METHOD FB_init : BOOL
VAR_INPUT
	bInitRetains : BOOL; // if TRUE, the retain variables are initialized (warm start / cold start)
	bInCopyCode : BOOL;  // if TRUE, the instance afterwards gets moved into the copy code (online change)
END_VAR
AddInput('ipSrcImage', ipSrcImage);
AddInput('ipTemplateImage', ipTemplateImage);
AddInput('fMatchThreshold', fMatchThreshold);
AddInput('nProjections', nProjections);
AddInput('eOptions', eOptions);
AddInput('nRotations', nRotations);
AddInput('fScaleFactor', fScaleFactor);
AddInput('eInterpolationType', eInterpolationType);
AddInput('hrPrev', hrPrev);
AddOutput('ipMatches', ipMatches);
AddOutput('ipMatchValues', ipMatchValues);
AddOutput('hresult',hresult);
END_METHOD

METHOD PUBLIC  Clone : I_Node
VAR
	pNode : POINTER TO Node_F_VN_FindTemplateWalshExp;
END_VAR
pNode := __NEW(Node_F_VN_FindTemplateWalshExp);
Clone := pNode^;
END_METHOD

METHOD PROTECTED OnExecute
hresult.Value := F_VN_FindTemplateWalshExp(
    ipSrcImage := ipSrcImage.Value,
    ipTemplateImage := ipTemplateImage.Value,
	ipMatches := ipMatches.Value,
	fMatchThreshold := fMatchThreshold.Value,
	nProjections := nProjections.Value,
	eOptions := eOptions.Value,
	nRotations := nRotations.Value,
	fScaleFactor := fScaleFactor.Value,
	eInterpolationType := eInterpolationType.Value,
	ipMatchValues := ipMatchValues.Value,
	hrPrev:= hrPrev.Value);
END_METHOD

METHOD PUBLIC PreExecutionCheck
VAR_INPUT
	Check : I_PreExecutionChecks;
END_VAR
Check.IsTrue(ipSrcImage.IsValid, 'ipSrcImage must contain an image');
Check.IsTrue(ipSrcImage.IsPixelDepth(8), 'ipSrcImage must be 8 or 32 bit pixel depth');
Check.IsTrue((ipSrcImage.HasChannelCount(1) OR ipSrcImage.HasChannelCount(3)), 'ipSrcImage must contain 1 or 3 channels');

Check.IsTrue((nRotations.Value = 1 OR nRotations.Value = 2 OR nRotations.Value = 4 OR nRotations.Value = 8 OR nRotations.Value = 16 OR nRotations.Value = 32), 'nRotations must be 1, 2, 4, 8, 16 or 32');
Check.IsTrue((fMatchThreshold.Value >= 0 AND fMatchThreshold.Value <= 1), 'Threshold must be between 0..1, 1.0 would be a perfect match');
Check.IsTrue(nProjections.Value <= 50, 'The soft limit of 50 has been reached');

Check.IsTrue(ipTemplateImage.IsValid, 'ipTemplateImage must contain an image');
Check.IsTrue(ImagesHaveMatchingPixelFormats(ipSrcImage.Value, ipTemplateImage.Value), 'ipTemplateImage must have same pixel depth as ipSrcImage');
Check.IsTrue(ImagesHaveMatchingChannels(ipSrcImage.Value, ipTemplateImage.Value), 'ipTemplateImage must have same amount of channels as ipSrcImage');
Check.IsTrue(IsTemplateImageSmallerThanSourceImage(ipSrcImage.Value, ipTemplateImage.Value), 'ipTemplateImage must be smaller than ipSrcImage');
END_METHOD

END_FUNCTION_BLOCK

// Nodes/Image Analysis/Object Detection/Node_F_VN_FindTemplateWalshExp_AngleRange
{attribute 'linkalways'} 
{attribute 'no_explicit_call' := 'This FB is a CLASS and must be accessed using methods or properties'}
{attribute 'enable_dynamic_creation'}
FUNCTION_BLOCK Node_F_VN_FindTemplateWalshExp_AngleRange EXTENDS VisionNode
VAR
    ipSrcImage : _ITcVnImage;
    ipTemplateImage : _ITcVnImage;
	ipMatches : _ITcVnContainer;
	fMatchThreshold : _REAL(0.1);
	nProjections : _UDINT(10);
	fStartAngle : _LREAL(0);
	fStopAngle : _LREAL(1);
	nAngles : _UDINT(1);
	eOptions : _ETcVnFindTemplateWalshOptions(ETcVnFindTemplateWalshOptions.TCVN_FTWO_NONE);
	fScaleFactor : _REAL(1);
	eInterpolationType : _ETcVnInterpolationType(ETcVnInterpolationType.TCVN_IT_AREA_BASED);
	ipMatchValues : _ITcVnContainer;
    hrPrev : _HRESULT(S_OK);
	hresult : _HRESULT(S_OK);
END_VAR

METHOD FB_init : BOOL
VAR_INPUT
	bInitRetains : BOOL; // if TRUE, the retain variables are initialized (warm start / cold start)
	bInCopyCode : BOOL;  // if TRUE, the instance afterwards gets moved into the copy code (online change)
END_VAR
AddInput('ipSrcImage', ipSrcImage);
AddInput('ipTemplateImage', ipTemplateImage);
AddInput('fMatchThreshold', fMatchThreshold);
AddInput('nProjections', nProjections);
AddInput('fStartAngle', fStartAngle);
AddInput('fStopAngle', fStopAngle);
AddInput('nAngles', nAngles);
AddInput('eOptions', eOptions);
AddInput('fScaleFactor', fScaleFactor);
AddInput('eInterpolationType', eInterpolationType);
AddInput('hrPrev', hrPrev);
AddOutput('ipMatches', ipMatches);
AddOutput('ipMatchValues', ipMatchValues);
AddOutput('hresult',hresult);
END_METHOD

METHOD PUBLIC  Clone : I_Node
VAR
	pNode : POINTER TO Node_F_VN_FindTemplateWalshExp_AngleRange;
END_VAR
pNode := __NEW(Node_F_VN_FindTemplateWalshExp_AngleRange);
Clone := pNode^;
END_METHOD

METHOD PROTECTED OnExecute
hresult.Value := F_VN_FindTemplateWalshExp_AngleRange(
    ipSrcImage := ipSrcImage.Value,
    ipTemplateImage := ipTemplateImage.Value,
	ipMatches := ipMatches.Value,
	fMatchThreshold := fMatchThreshold.Value,
	nProjections := nProjections.Value,
	fStartAngle := fStartAngle.Value,
	fStopAngle := fStopAngle.Value,
	nAngles := nAngles.Value,
	eOptions := eOptions.Value,
	fScaleFactor := fScaleFactor.Value,
	eInterpolationType := eInterpolationType.Value,
	ipMatchValues := ipMatchValues.Value,
	hrPrev:= hrPrev.Value);
END_METHOD

METHOD PUBLIC PreExecutionCheck
VAR_INPUT
	Check : I_PreExecutionChecks;
END_VAR
Check.IsTrue(ipSrcImage.IsValid, 'ipSrcImage must contain an image');
Check.IsTrue(ipSrcImage.IsPixelDepth(8), 'ipSrcImage must be 8 or 32 bit pixel depth');
Check.IsTrue((ipSrcImage.HasChannelCount(1) OR ipSrcImage.HasChannelCount(3)), 'ipSrcImage must contain 1 or 3 channels');

Check.IsTrue((fMatchThreshold.Value >= 0 AND fMatchThreshold.Value <= 1), 'Threshold must be between 0..1, 1.0 would be a perfect match');
Check.IsTrue(nProjections.Value <= 50, 'The soft limit of 50 has been reached');

Check.IsTrue(ipTemplateImage.IsValid, 'ipTemplateImage must contain an image');
Check.IsTrue(ImagesHaveMatchingPixelFormats(ipSrcImage.Value, ipTemplateImage.Value), 'ipTemplateImage must have same pixel depth as ipSrcImage');
Check.IsTrue(ImagesHaveMatchingChannels(ipSrcImage.Value, ipTemplateImage.Value), 'ipTemplateImage must have same amount of channels as ipSrcImage');
Check.IsTrue(IsTemplateImageSmallerThanSourceImage(ipSrcImage.Value, ipTemplateImage.Value), 'ipTemplateImage must be smaller than ipSrcImage');
END_METHOD

END_FUNCTION_BLOCK

// Nodes/Image Analysis/Object Detection/Node_F_VN_HoughCircles
{attribute 'linkalways'} 
{attribute 'no_explicit_call' := 'This FB is a CLASS and must be accessed using methods or properties'}
{attribute 'enable_dynamic_creation'}
FUNCTION_BLOCK Node_F_VN_HoughCircles EXTENDS VisionNode
VAR
    ipSrcImage : _ITcVnImage;
    ipCircles : _ITcVnContainer;
    fInvAccuRatio : _LREAL(1.0);
    fMinDist : _LREAL(1.0);
    hrPrev : _HRESULT(S_OK);
	hresult : _HRESULT(S_OK);
END_VAR

METHOD FB_init : BOOL
VAR_INPUT
	bInitRetains : BOOL; // if TRUE, the retain variables are initialized (warm start / cold start)
	bInCopyCode : BOOL;  // if TRUE, the instance afterwards gets moved into the copy code (online change)
END_VAR
AddInput('ipSrcImage', ipSrcImage);
AddParameter('fInvAccuRatio', fInvAccuRatio);
AddParameter('fMinDist', fMinDist);
AddInput('hrPrev', hrPrev);
AddOutput('ipCircles', ipCircles);
AddOutput('hresult', hresult);
END_METHOD

METHOD PUBLIC  Clone : I_Node
VAR
	pNode : POINTER TO Node_F_VN_HoughCircles;
END_VAR
pNode := __NEW(Node_F_VN_HoughCircles);
Clone := pNode^;
END_METHOD

METHOD PROTECTED OnExecute
hresult.Value := F_VN_HoughCircles(
	ipSrcImage := ipSrcImage.Value,
    ipCircles := ipCircles.Value,
    fInvAccuRatio := fInvAccuRatio.Value,
    fMinDist := fMinDist.Value,
	hrPrev:= hrPrev.Value);
END_METHOD

METHOD PUBLIC PreExecutionCheck
VAR_INPUT
	Check : I_PreExecutionChecks;
END_VAR
Check.IsTrue(ipSrcImage.IsValid, 'ipSrcImage must contain an image');
Check.IsTrue(ipSrcImage.IsElementType(ETcVnElementType.TCVN_ET_USINT), 'ipSrcImage must be usint');
Check.IsTrue(ipSrcImage.HasChannelCount(1), 'ipSrcImage must contain 1 channel');
Check.IsTrue((fInvAccuRatio.Value > 0), 'fInvAccuRatio must be greater than 0');
Check.IsTrue((fMinDist.Value > 0), 'fMinDist must be greater than 0');
END_METHOD

END_FUNCTION_BLOCK

// Nodes/Image Analysis/Object Detection/Node_F_VN_HoughCirclesExp
{attribute 'linkalways'} 
{attribute 'no_explicit_call' := 'This FB is a CLASS and must be accessed using methods or properties'}
{attribute 'enable_dynamic_creation'}
FUNCTION_BLOCK Node_F_VN_HoughCirclesExp EXTENDS VisionNode
VAR
    ipSrcImage : _ITcVnImage;
    ipCircles : _ITcVnContainer;
    fInvAccuRatio : _LREAL(1.0);
    fMinDist : _LREAL(1.0);
	eHoughMethod : _ETcVnHoughMethod(ETcVnHoughMethod.TCVN_HM_GRADIENT);
    fParam1 : _LREAL(0.0);
	fParam2 : _LREAL(0.0);
	nMinRadius : _UDINT(0);
	nMaxRadius : _UDINT(0);
	hrPrev : _HRESULT(S_OK);
	hresult : _HRESULT(S_OK);
END_VAR

METHOD FB_init : BOOL
VAR_INPUT
	bInitRetains : BOOL; // if TRUE, the retain variables are initialized (warm start / cold start)
	bInCopyCode : BOOL;  // if TRUE, the instance afterwards gets moved into the copy code (online change)
END_VAR
AddInput('ipSrcImage', ipSrcImage);
AddParameter('fInvAccuRatio', fInvAccuRatio);
AddParameter('fMinDist', fMinDist);
AddParameter('eHoughMethod', eHoughMethod);
AddParameter('fParam1', fParam1);
AddParameter('fParam2', fParam2);
AddParameter('nMinRadius', nMinRadius);
AddParameter('nMaxRadius', nMaxRadius);
AddInput('hrPrev', hrPrev);
AddOutput('ipCircles', ipCircles);
AddOutput('hresult', hresult);
END_METHOD

METHOD PUBLIC  Clone : I_Node
VAR
	pNode : POINTER TO Node_F_VN_HoughCirclesExp;
END_VAR
pNode := __NEW(Node_F_VN_HoughCirclesExp);
Clone := pNode^;
END_METHOD

METHOD PROTECTED OnExecute
hresult.Value := F_VN_HoughCirclesExp(
	ipSrcImage := ipSrcImage.Value,
    ipCircles := ipCircles.Value,
    fInvAccuRatio := fInvAccuRatio.Value,
    fMinDist := fMinDist.Value,
	eHoughMethod := eHoughMethod.Value,
	fParam1 := fParam1.Value,
	fParam2 := fParam2.Value,
	nMinRadius := nMinRadius.Value,
	nMaxRadius := nMaxRadius.Value,
	hrPrev:= hrPrev.Value);
END_METHOD

METHOD PUBLIC PreExecutionCheck
VAR_INPUT
	Check : I_PreExecutionChecks;
END_VAR
Check.IsTrue(ipSrcImage.IsValid, 'ipSrcImage must contain an image');
Check.IsTrue(ipSrcImage.IsElementType(ETcVnElementType.TCVN_ET_USINT), 'ipSrcImage must be usint');
Check.IsTrue(ipSrcImage.HasChannelCount(1), 'ipSrcImage must contain 1 channel');
Check.IsTrue((fInvAccuRatio.Value > 0), 'fInvAccuRatio must be greater than 0');
Check.IsTrue((fMinDist.Value > 0), 'fMinDist must be greater than 0');

Check.IsTrue(
    (eHoughMethod.Value = ETcVnHoughMethod.TCVN_HM_GRADIENT) OR
    (eHoughMethod.Value = ETcVnHoughMethod.TCVN_HM_GRADIENT_ALT),
    'eHoughMethod must be GRADIENT or GRADIENT_ALT');
	
	
IF (eHoughMethod.Value = ETcVnHoughMethod.TCVN_HM_GRADIENT_ALT) THEN
    Check.IsTrue((fParam2.Value > 0) AND (fParam2.Value < 1),
        'fParam2 (circle perfectness) must be > 0 and < 1 for GRADIENT_ALT');
ELSE
    Check.IsTrue((fParam2.Value > 0),
        'fParam2 (accumulator threshold) must be > 0 for GRADIENT');
END_IF

IF (nMaxRadius.Value > 0) THEN
    Check.IsTrue((nMaxRadius.Value >= nMinRadius.Value),
        'nMaxRadius must be >= nMinRadius when non-zero');
END_IF
END_METHOD

END_FUNCTION_BLOCK

// Nodes/Image Analysis/Object Detection/Node_F_VN_HoughLines
{attribute 'linkalways'} 
{attribute 'no_explicit_call' := 'This FB is a CLASS and must be accessed using methods or properties'}
{attribute 'enable_dynamic_creation'}
FUNCTION_BLOCK Node_F_VN_HoughLines EXTENDS VisionNode
VAR
    ipSrcImage : _ITcVnImage;
    ipLines : _ITcVnContainer;
    fDistRes : _LREAL(1.0);
    fAngleRes : _LREAL(1.0);
    nAccuThreshold : _UDINT(0);
    hrPrev : _HRESULT(S_OK);
	hresult : _HRESULT(S_OK);
END_VAR

METHOD FB_init : BOOL
VAR_INPUT
	bInitRetains : BOOL; // if TRUE, the retain variables are initialized (warm start / cold start)
	bInCopyCode : BOOL;  // if TRUE, the instance afterwards gets moved into the copy code (online change)
END_VAR
AddInput('ipSrcImage', ipSrcImage);
AddParameter('fDistRes', fDistRes);
AddParameter('fAngleRes', fAngleRes);
AddParameter('nAccuThreshold', nAccuThreshold);
AddInput('hrPrev', hrPrev);
AddOutput('ipLines', ipLines);
AddOutput('hresult', hresult);
END_METHOD

METHOD PUBLIC  Clone : I_Node
VAR
	pNode : POINTER TO Node_F_VN_HoughLines;
END_VAR
pNode := __NEW(Node_F_VN_HoughLines);
Clone := pNode^;
END_METHOD

METHOD PROTECTED OnExecute
hresult.Value := F_VN_HoughLines(
	ipSrcImage := ipSrcImage.Value,
    ipLines := ipLines.Value,
    fDistRes := fDistRes.Value,
    fAngleRes := fAngleRes.Value,
    nAccuThreshold := nAccuThreshold.Value,
	hrPrev:= hrPrev.Value);
END_METHOD

METHOD PUBLIC PreExecutionCheck
VAR_INPUT
	Check : I_PreExecutionChecks;
END_VAR
Check.IsTrue(ipSrcImage.IsValid, 'ipSrcImage must contain an image');
Check.IsTrue(ipSrcImage.IsPixelDepth(8), 'ipSrcImage must be 8 bit pixel depth');
Check.IsTrue(ipSrcImage.HasChannelCount(1), 'ipSrcImage must contain 1 channel');
Check.IsTrue((fDistRes.Value > 0), 'fDistRes must be greater than 0');
Check.IsTrue((fAngleRes.Value > 0), 'fAngleRes must be greater than 0');
END_METHOD

END_FUNCTION_BLOCK

// Nodes/Image Analysis/Object Detection/Node_F_VN_HoughLinesP
{attribute 'linkalways'} 
{attribute 'no_explicit_call' := 'This FB is a CLASS and must be accessed using methods or properties'}
{attribute 'enable_dynamic_creation'}
FUNCTION_BLOCK Node_F_VN_HoughLinesP EXTENDS VisionNode
VAR
    ipSrcImage : _ITcVnImage;
    ipLines : _ITcVnContainer;
    fDistRes : _LREAL(1.0);
    fAngleRes : _LREAL(1.0);
    nAccuThreshold : _UDINT(0);
    hrPrev : _HRESULT(S_OK);
	hresult : _HRESULT(S_OK);
END_VAR

METHOD FB_init : BOOL
VAR_INPUT
	bInitRetains : BOOL; // if TRUE, the retain variables are initialized (warm start / cold start)
	bInCopyCode : BOOL;  // if TRUE, the instance afterwards gets moved into the copy code (online change)
END_VAR
AddInput('ipSrcImage', ipSrcImage);
AddParameter('fDistRes', fDistRes);
AddParameter('fAngleRes', fAngleRes);
AddParameter('nAccuThreshold', nAccuThreshold);
AddInput('hrPrev', hrPrev);
AddOutput('ipLines', ipLines);
AddOutput('hresult', hresult);
END_METHOD

METHOD PUBLIC  Clone : I_Node
VAR
	pNode : POINTER TO Node_F_VN_HoughLinesP;
END_VAR
pNode := __NEW(Node_F_VN_HoughLinesP);
Clone := pNode^;
END_METHOD

METHOD PROTECTED OnExecute
hresult.Value := F_VN_HoughLinesP(
	ipSrcImage := ipSrcImage.Value,
    ipLines := ipLines.Value,
    fDistRes := fDistRes.Value,
    fAngleRes := fAngleRes.Value,
    nAccuThreshold := nAccuThreshold.Value,
	hrPrev:= hrPrev.Value);
END_METHOD

METHOD PUBLIC PreExecutionCheck
VAR_INPUT
	Check : I_PreExecutionChecks;
END_VAR
Check.IsTrue(ipSrcImage.IsValid, 'ipSrcImage must contain an image');
Check.IsTrue(ipSrcImage.IsPixelDepth(8), 'ipSrcImage must be 8 bit pixel depth');
Check.IsTrue(ipSrcImage.HasChannelCount(1), 'ipSrcImage must contain 1 channel');
Check.IsTrue((fDistRes.Value > 0), 'fDistRes must be greater than 0');
Check.IsTrue((fAngleRes.Value > 0), 'fAngleRes must be greater than 0');
END_METHOD

END_FUNCTION_BLOCK

// Nodes/Image Analysis/Object Detection/Node_F_VN_HoughLinesPExp
{attribute 'linkalways'} 
{attribute 'no_explicit_call' := 'This FB is a CLASS and must be accessed using methods or properties'}
{attribute 'enable_dynamic_creation'}
FUNCTION_BLOCK Node_F_VN_HoughLinesPExp EXTENDS VisionNode
VAR
    ipSrcImage : _ITcVnImage;
    ipLines : _ITcVnContainer;
    fDistRes : _LREAL(1.0);
    fAngleRes : _LREAL(1.0);
    nAccuThreshold : _UDINT(0);
    fMinLineLength : _LREAL(0.0);
    fMaxLineGap : _LREAL(0.0);
    hrPrev : _HRESULT(S_OK);
	hresult : _HRESULT(S_OK);
END_VAR

METHOD FB_init : BOOL
VAR_INPUT
	bInitRetains : BOOL; // if TRUE, the retain variables are initialized (warm start / cold start)
	bInCopyCode : BOOL;  // if TRUE, the instance afterwards gets moved into the copy code (online change)
END_VAR
AddInput('ipSrcImage', ipSrcImage);
AddParameter('fDistRes', fDistRes);
AddParameter('fAngleRes', fAngleRes);
AddParameter('nAccuThreshold', nAccuThreshold);
AddParameter('fMinLineLength', fMinLineLength);
AddParameter('fMaxLineGap', fMaxLineGap);
AddInput('hrPrev', hrPrev);
AddOutput('ipLines', ipLines);
AddOutput('hresult', hresult);
END_METHOD

METHOD PUBLIC  Clone : I_Node
VAR
	pNode : POINTER TO Node_F_VN_HoughLinesPExp;
END_VAR
pNode := __NEW(Node_F_VN_HoughLinesPExp);
Clone := pNode^;
END_METHOD

METHOD PROTECTED OnExecute
hresult.Value := F_VN_HoughLinesPExp(
	ipSrcImage := ipSrcImage.Value,
    ipLines := ipLines.Value,
    fDistRes := fDistRes.Value,
    fAngleRes := fAngleRes.Value,
    nAccuThreshold := nAccuThreshold.Value,
    fMinLineLength := fMinLineLength.Value,
    fMaxLineGap := fMaxLineGap.Value,
	hrPrev:= hrPrev.Value);
END_METHOD

METHOD PUBLIC PreExecutionCheck
VAR_INPUT
	Check : I_PreExecutionChecks;
END_VAR
Check.IsTrue(ipSrcImage.IsValid, 'ipSrcImage must contain an image');
Check.IsTrue(ipSrcImage.IsPixelDepth(8), 'ipSrcImage must be 8 bit pixel depth');
Check.IsTrue(ipSrcImage.HasChannelCount(1), 'ipSrcImage must contain 1 channel');
Check.IsTrue((fDistRes.Value > 0), 'fDistRes must be greater than 0');
Check.IsTrue((fAngleRes.Value > 0), 'fAngleRes must be greater than 0');
END_METHOD

END_FUNCTION_BLOCK

// Nodes/Image Analysis/Object Detection/Node_F_VN_MatchImageHuMoments
{attribute 'linkalways'} 
{attribute 'no_explicit_call' := 'This FB is a CLASS and must be accessed using methods or properties'}
{attribute 'enable_dynamic_creation'}
FUNCTION_BLOCK Node_F_VN_MatchImageHuMoments EXTENDS VisionNode
VAR
    ipImage1 : _ITcVnImage;
    ipImage2 : _ITcVnImage;
    eComparisonMethod : _ETcVnContoursMatchComparisonMethod(ETcVnContoursMatchComparisonMethod.TCVN_CMCM_CONTOURS_MATCH_I1);
    fDissimilarity : _LREAL(0.0);
    hrPrev : _HRESULT(S_OK);
	hresult : _HRESULT(S_OK);
END_VAR

METHOD FB_init : BOOL
VAR_INPUT
	bInitRetains : BOOL; // if TRUE, the retain variables are initialized (warm start / cold start)
	bInCopyCode : BOOL;  // if TRUE, the instance afterwards gets moved into the copy code (online change)
END_VAR
AddInput('ipImage1', ipImage1);
AddInput('ipImage2', ipImage2);
AddParameter('eComparisonMethod', eComparisonMethod);
AddInput('hrPrev', hrPrev);
AddOutput('fDissimilarity', fDissimilarity);
AddOutput('hresult', hresult);
END_METHOD

METHOD PUBLIC  Clone : I_Node
VAR
	pNode : POINTER TO Node_F_VN_MatchImageHuMoments;
END_VAR
pNode := __NEW(Node_F_VN_MatchImageHuMoments);
Clone := pNode^;
END_METHOD

METHOD PROTECTED OnExecute
hresult.Value := F_VN_MatchImageHuMoments(
	ipImage1 := ipImage1.Value,
    ipImage2 := ipImage2.Value,
    eComparisonMethod := eComparisonMethod.Value,
    fDissimilarity := fDissimilarity.Value,
	hrPrev:= hrPrev.Value);
END_METHOD

METHOD PUBLIC PreExecutionCheck
VAR_INPUT
	Check : I_PreExecutionChecks;
END_VAR
Check.IsTrue(ipImage1.IsValid, 'ipImage1 must contain an image');
Check.IsTrue(ipImage1.HasChannelCount(1), 'ipImage1 must contain 1 channel');
Check.IsTrue(ipImage2.IsValid, 'ipImage2 must contain an image');
Check.IsTrue(ipImage2.HasChannelCount(1), 'ipImage2 must contain 1 channel');
END_METHOD

END_FUNCTION_BLOCK

// Nodes/Image Analysis/Object Detection/Node_F_VN_MatchTemplate
{attribute 'linkalways'} 
{attribute 'no_explicit_call' := 'This FB is a CLASS and must be accessed using methods or properties'}
{attribute 'enable_dynamic_creation'}
FUNCTION_BLOCK Node_F_VN_MatchTemplate EXTENDS VisionNode
VAR
    ipSrcImage : _ITcVnImage;
    ipTemplateImage : _ITcVnImage;
    ipResultImage : _ITcVnImage;
    hrPrev : _HRESULT(S_OK);
	hresult : _HRESULT(S_OK);
END_VAR

METHOD FB_init : BOOL
VAR_INPUT
	bInitRetains : BOOL; // if TRUE, the retain variables are initialized (warm start / cold start)
	bInCopyCode : BOOL;  // if TRUE, the instance afterwards gets moved into the copy code (online change)
END_VAR
AddInput('ipSrcImage', ipSrcImage);
AddInput('ipTemplateImage', ipTemplateImage);
AddInput('hrPrev', hrPrev);
AddOutput('ipResultImage', ipResultImage);
AddOutput('hresult',hresult);
END_METHOD

METHOD PUBLIC  Clone : I_Node
VAR
	pNode : POINTER TO Node_F_VN_MatchTemplate;
END_VAR
pNode := __NEW(Node_F_VN_MatchTemplate);
Clone := pNode^;
END_METHOD

METHOD PROTECTED OnExecute
hresult.Value := F_VN_MatchTemplate(
    ipSrcImage := ipSrcImage.Value,
    ipTemplateImage := ipTemplateImage.Value,
	ipResultImage := ipResultImage.Value,
	hrPrev:= hrPrev.Value);
END_METHOD

METHOD PUBLIC PreExecutionCheck
VAR_INPUT
	Check : I_PreExecutionChecks;
END_VAR
Check.IsTrue(ipSrcImage.IsValid, 'ipSrcImage must contain an image');
Check.IsTrue((ipSrcImage.IsPixelDepth(8) OR ipSrcImage.IsPixelDepth(32)), 'ipSrcImage must be 8 or 32 bit pixel depth');
Check.IsTrue((ipSrcImage.HasChannelCount(1) OR ipSrcImage.HasChannelCount(3)), 'ipSrcImage must contain 1 or 3 channels');

Check.IsTrue(ipTemplateImage.IsValid, 'ipTemplateImage must contain an image');
Check.IsTrue(ImagesHaveMatchingPixelFormats(ipSrcImage.Value, ipTemplateImage.Value), 'ipTemplateImage must have same pixel depth as ipSrcImage');
Check.IsTrue(ImagesHaveMatchingChannels(ipSrcImage.Value, ipTemplateImage.Value), 'ipTemplateImage must have same amount of channels as ipSrcImage');
Check.IsTrue(IsTemplateImageSmallerThanSourceImage(ipSrcImage.Value, ipTemplateImage.Value), 'ipTemplateImage must be smaller than ipSrcImage');
END_METHOD

END_FUNCTION_BLOCK

// Nodes/Image Analysis/Object Detection/Node_F_VN_MatchTemplateAndEvaluate
{attribute 'linkalways'} 
{attribute 'no_explicit_call' := 'This FB is a CLASS and must be accessed using methods or properties'}
{attribute 'enable_dynamic_creation'}
FUNCTION_BLOCK Node_F_VN_MatchTemplateAndEvaluate EXTENDS VisionNode
VAR
    ipSrcImage : _ITcVnImage;
    ipTemplateImage : _ITcVnImage;
    ipMatches : _ITcVnContainer;
    fMatchThreshold : _REAL(0.0);
    hrPrev : _HRESULT(S_OK);
	hresult : _HRESULT(S_OK);
END_VAR

METHOD FB_init : BOOL
VAR_INPUT
	bInitRetains : BOOL; // if TRUE, the retain variables are initialized (warm start / cold start)
	bInCopyCode : BOOL;  // if TRUE, the instance afterwards gets moved into the copy code (online change)
END_VAR
AddInput('ipSrcImage', ipSrcImage);
AddInput('ipTemplateImage', ipTemplateImage);
AddParameter('fMatchThreshold', fMatchThreshold);
AddInput('hrPrev', hrPrev);
AddOutput('ipMatches', ipMatches);
AddOutput('hresult',hresult);
END_METHOD

METHOD PUBLIC  Clone : I_Node
VAR
	pNode : POINTER TO Node_F_VN_MatchTemplateAndEvaluate;
END_VAR
pNode := __NEW(Node_F_VN_MatchTemplateAndEvaluate);
Clone := pNode^;
END_METHOD

METHOD PROTECTED OnExecute
hresult.Value := F_VN_MatchTemplateAndEvaluate(
    ipSrcImage := ipSrcImage.Value,
    ipTemplateImage := ipTemplateImage.Value,
	ipMatches := ipMatches.Value,
    fMatchThreshold := fMatchThreshold.Value,
	hrPrev:= hrPrev.Value);
END_METHOD

METHOD PUBLIC PreExecutionCheck
VAR_INPUT
	Check : I_PreExecutionChecks;
END_VAR
Check.IsTrue(ipSrcImage.IsValid, 'ipSrcImage must contain an image');
Check.IsTrue((ipSrcImage.IsPixelDepth(8) OR ipSrcImage.IsPixelDepth(32)), 'ipSrcImage must be 8 or 32 bit pixel depth');
Check.IsTrue((ipSrcImage.HasChannelCount(1) OR ipSrcImage.HasChannelCount(3)), 'ipSrcImage must contain 1 or 3 channels');

Check.IsTrue(ipTemplateImage.IsValid, 'ipTemplateImage must contain an image');
Check.IsTrue(ImagesHaveMatchingPixelFormats(ipSrcImage.Value, ipTemplateImage.Value), 'ipTemplateImage must have same pixel depth ipSrcImage');
Check.IsTrue(ImagesHaveMatchingChannels(ipSrcImage.Value, ipTemplateImage.Value), 'ipTemplateImage must have same amount of channels as ipSrcImage');
Check.IsTrue(IsTemplateImageSmallerThanSourceImage(ipSrcImage.Value, ipTemplateImage.Value), 'ipTemplateImage must be smaller than ipSrcImage');

Check.IsTrue((fMatchThreshold.Value >= 0.0) AND (fMatchThreshold.Value <= 1.0), 'fMatchThreshold must be between 0 and 1');
END_METHOD

END_FUNCTION_BLOCK

// Nodes/Image Analysis/Object Detection/Node_F_VN_MatchTemplateAndEvaluateExp
{attribute 'linkalways'}
{attribute 'no_explicit_call' := 'This FB is a CLASS and must be accessed using methods or properties'}
{attribute 'enable_dynamic_creation'}
FUNCTION_BLOCK Node_F_VN_MatchTemplateAndEvaluateExp EXTENDS VisionNode
VAR
    ipSrcImage : _ITcVnImage;
    ipTemplateImage : _ITcVnImage;
    ipMatches : _ITcVnContainer;
    fMatchThreshold : _REAL(0.0);
    eMatchMethod : _ETcVnTemplateMatchMethod(ETcVnTemplateMatchMethod.TCVN_TMM_CCORR_NORMED);
    ipTemplateMask : _ITcVnImage;
    fScaleFactor : _REAL(1);
    eInterpolationType : _ETcVnInterpolationType(ETcVnInterpolationType.TCVN_IT_BILINEAR);
    ipMatchValues : _ITcVnContainer;
    hrPrev : _HRESULT(S_OK);
    hresult : _HRESULT(S_OK);
END_VAR

METHOD FB_init : BOOL
VAR_INPUT
    bInitRetains : BOOL;
    bInCopyCode : BOOL;
END_VAR
AddInput('ipSrcImage', ipSrcImage);
AddInput('ipTemplateImage', ipTemplateImage);
AddOutput('ipMatches', ipMatches);
AddParameter('fMatchThreshold', fMatchThreshold);
AddParameter('eMatchMethod', eMatchMethod);
AddInput('ipTemplateMask', ipTemplateMask);
AddParameter('fScaleFactor', fScaleFactor);
AddParameter('eInterpolationType', eInterpolationType);
AddOutput('ipMatchValues', ipMatchValues);
AddInput('hrPrev', hrPrev);
AddOutput('hresult', hresult);
END_METHOD

METHOD PUBLIC Clone : I_Node
VAR
    pNode : POINTER TO Node_F_VN_MatchTemplateAndEvaluateExp;
END_VAR
pNode := __NEW(Node_F_VN_MatchTemplateAndEvaluateExp);
Clone := pNode^;
END_METHOD

METHOD PROTECTED OnExecute
hresult.Value := F_VN_MatchTemplateAndEvaluateExp(
    ipSrcImage := ipSrcImage.Value,
    ipTemplateImage := ipTemplateImage.Value,
    ipMatches := ipMatches.Value,
    fMatchThreshold := fMatchThreshold.Value,
    eMatchMethod := eMatchMethod.Value,
    ipTemplateMask := ipTemplateMask.Value,
    fScaleFactor := fScaleFactor.Value,
    eInterpolationType := eInterpolationType.Value,
    ipMatchValues := ipMatchValues.Value,
    hrPrev := hrPrev.Value);
END_METHOD

METHOD PUBLIC PreExecutionCheck
VAR_INPUT
    Check : I_PreExecutionChecks;
END_VAR
Check.IsTrue(ipSrcImage.IsValid, 'ipSrcImage must contain an image');
Check.IsTrue(ipSrcImage.IsElementType(ETcVnElementType.TCVN_ET_USINT) OR ipSrcImage.IsElementType(ETcVnElementType.TCVN_ET_REAL), 'ipSrcImage must contain USINT or REAL elements');
Check.IsTrue(ipSrcImage.HasChannelCount(1) OR ipSrcImage.HasChannelCount(3), 'ipSrcImage must contain 1 or 3 channels');
Check.IsTrue(ipTemplateImage.IsValid, 'ipTemplateImage must contain an image');
Check.IsTrue(ImagesHaveMatchingPixelFormats(ipSrcImage.Value, ipTemplateImage.Value), 'Source and template must have matching pixel formats');
Check.IsTrue(IsTemplateImageSmallerThanSourceImage(ipSrcImage.Value, ipTemplateImage.Value), 'Template width and height must be smaller than the source');
IF ipTemplateMask.Value <> 0 THEN
    Check.IsTrue(ipTemplateMask.IsValid, 'ipTemplateMask must contain an image when connected');
    Check.IsTrue(ImagesHaveMatchingPixelFormats(ipTemplateImage.Value, ipTemplateMask.Value), 'Template and mask must have matching pixel formats');
    Check.IsTrue(IsImage1SizeEqualToImage2Size(ipTemplateImage.Value, ipTemplateMask.Value), 'Template and mask must have matching dimensions');
END_IF
Check.IsTrue((eMatchMethod.Value = ETcVnTemplateMatchMethod.TCVN_TMM_SQDIFF) OR
             (eMatchMethod.Value = ETcVnTemplateMatchMethod.TCVN_TMM_SQDIFF_NORMED) OR
             (eMatchMethod.Value = ETcVnTemplateMatchMethod.TCVN_TMM_CCORR) OR
             (eMatchMethod.Value = ETcVnTemplateMatchMethod.TCVN_TMM_CCORR_NORMED) OR
             (eMatchMethod.Value = ETcVnTemplateMatchMethod.TCVN_TMM_CCOEFF) OR
             (eMatchMethod.Value = ETcVnTemplateMatchMethod.TCVN_TMM_CCOEFF_NORMED), 'Unsupported eMatchMethod');
Check.IsTrue((fScaleFactor.Value > 0.0) AND (fScaleFactor.Value <= 1.0), 'Scale factor must be greater than 0 and at most 1');
IF (eMatchMethod.Value = ETcVnTemplateMatchMethod.TCVN_TMM_SQDIFF_NORMED) OR
   (eMatchMethod.Value = ETcVnTemplateMatchMethod.TCVN_TMM_CCORR_NORMED) OR
   (eMatchMethod.Value = ETcVnTemplateMatchMethod.TCVN_TMM_CCOEFF_NORMED) THEN
    Check.IsTrue((fMatchThreshold.Value >= 0.0) AND (fMatchThreshold.Value <= 1.0), 'Normalized match threshold must be between 0 and 1');
END_IF
END_METHOD

END_FUNCTION_BLOCK

// Nodes/Image Analysis/Object Detection/Node_F_VN_MatchTemplateExp
{attribute 'linkalways'}
{attribute 'no_explicit_call' := 'This FB is a CLASS and must be accessed using methods or properties'}
{attribute 'enable_dynamic_creation'}
FUNCTION_BLOCK Node_F_VN_MatchTemplateExp EXTENDS VisionNode
VAR
    ipSrcImage : _ITcVnImage;
    ipTemplateImage : _ITcVnImage;
    ipResultImage : _ITcVnImage;
    eMatchMethod : _ETcVnTemplateMatchMethod(ETcVnTemplateMatchMethod.TCVN_TMM_CCORR_NORMED);
    ipTemplateMask : _ITcVnImage;
    hrPrev : _HRESULT(S_OK);
    hresult : _HRESULT(S_OK);
END_VAR

METHOD FB_init : BOOL
VAR_INPUT
    bInitRetains : BOOL;
    bInCopyCode : BOOL;
END_VAR
AddInput('ipSrcImage', ipSrcImage);
AddInput('ipTemplateImage', ipTemplateImage);
AddOutput('ipResultImage', ipResultImage);
AddParameter('eMatchMethod', eMatchMethod);
AddInput('ipTemplateMask', ipTemplateMask);
AddInput('hrPrev', hrPrev);
AddOutput('hresult', hresult);
END_METHOD

METHOD PUBLIC Clone : I_Node
VAR
    pNode : POINTER TO Node_F_VN_MatchTemplateExp;
END_VAR
pNode := __NEW(Node_F_VN_MatchTemplateExp);
Clone := pNode^;
END_METHOD

METHOD PROTECTED OnExecute
hresult.Value := F_VN_MatchTemplateExp(
    ipSrcImage := ipSrcImage.Value,
    ipTemplateImage := ipTemplateImage.Value,
    ipResultImage := ipResultImage.Value,
    eMatchMethod := eMatchMethod.Value,
    ipTemplateMask := ipTemplateMask.Value,
    hrPrev := hrPrev.Value);
END_METHOD

METHOD PUBLIC PreExecutionCheck
VAR_INPUT
    Check : I_PreExecutionChecks;
END_VAR
Check.IsTrue(ipSrcImage.IsValid, 'ipSrcImage must contain an image');
Check.IsTrue(ipSrcImage.IsElementType(ETcVnElementType.TCVN_ET_USINT) OR ipSrcImage.IsElementType(ETcVnElementType.TCVN_ET_REAL), 'ipSrcImage must contain USINT or REAL elements');
Check.IsTrue(ipSrcImage.HasChannelCount(1) OR ipSrcImage.HasChannelCount(3), 'ipSrcImage must contain 1 or 3 channels');
Check.IsTrue(ipTemplateImage.IsValid, 'ipTemplateImage must contain an image');
Check.IsTrue(ImagesHaveMatchingPixelFormats(ipSrcImage.Value, ipTemplateImage.Value), 'Source and template must have matching pixel formats');
Check.IsTrue(IsTemplateImageSmallerThanSourceImage(ipSrcImage.Value, ipTemplateImage.Value), 'Template width and height must be smaller than the source');
IF ipTemplateMask.Value <> 0 THEN
    Check.IsTrue(ipTemplateMask.IsValid, 'ipTemplateMask must contain an image when connected');
    Check.IsTrue(ImagesHaveMatchingPixelFormats(ipTemplateImage.Value, ipTemplateMask.Value), 'Template and mask must have matching pixel formats');
    Check.IsTrue(IsImage1SizeEqualToImage2Size(ipTemplateImage.Value, ipTemplateMask.Value), 'Template and mask must have matching dimensions');
END_IF
Check.IsTrue((eMatchMethod.Value = ETcVnTemplateMatchMethod.TCVN_TMM_SQDIFF) OR
             (eMatchMethod.Value = ETcVnTemplateMatchMethod.TCVN_TMM_SQDIFF_NORMED) OR
             (eMatchMethod.Value = ETcVnTemplateMatchMethod.TCVN_TMM_CCORR) OR
             (eMatchMethod.Value = ETcVnTemplateMatchMethod.TCVN_TMM_CCORR_NORMED) OR
             (eMatchMethod.Value = ETcVnTemplateMatchMethod.TCVN_TMM_CCOEFF) OR
             (eMatchMethod.Value = ETcVnTemplateMatchMethod.TCVN_TMM_CCOEFF_NORMED), 'Unsupported eMatchMethod');
END_METHOD

END_FUNCTION_BLOCK

// Nodes/Image Analysis/Object Detection/Node_F_VN_MatchTemplateWalsh
{attribute 'linkalways'} 
{attribute 'no_explicit_call' := 'This FB is a CLASS and must be accessed using methods or properties'}
{attribute 'enable_dynamic_creation'}
FUNCTION_BLOCK Node_F_VN_MatchTemplateWalsh EXTENDS VisionNode
VAR
    ipSrcImage : _ITcVnImage;
    ipTemplateImage : _ITcVnImage;
	nProjections : _UDINT(10);
    ipResultImage : _ITcVnImage;
    hrPrev : _HRESULT(S_OK);
	hresult : _HRESULT(S_OK);
END_VAR

METHOD FB_init : BOOL
VAR_INPUT
	bInitRetains : BOOL; // if TRUE, the retain variables are initialized (warm start / cold start)
	bInCopyCode : BOOL;  // if TRUE, the instance afterwards gets moved into the copy code (online change)
END_VAR
AddInput('ipSrcImage', ipSrcImage);
AddInput('ipTemplateImage', ipTemplateImage);
AddInput('nProjections', nProjections);
AddInput('hrPrev', hrPrev);
AddOutput('ipResultImage', ipResultImage);
AddOutput('hresult',hresult);
END_METHOD

METHOD PUBLIC  Clone : I_Node
VAR
	pNode : POINTER TO Node_F_VN_MatchTemplateWalsh;
END_VAR
pNode := __NEW(Node_F_VN_MatchTemplateWalsh);
Clone := pNode^;
END_METHOD

METHOD PROTECTED OnExecute
hresult.Value := F_VN_MatchTemplateWalsh(
    ipSrcImage := ipSrcImage.Value,
    ipTemplateImage := ipTemplateImage.Value,
	ipResultImage := ipResultImage.Value,
	nProjections := nProjections.Value,
	hrPrev:= hrPrev.Value);
END_METHOD

METHOD PUBLIC PreExecutionCheck
VAR_INPUT
	Check : I_PreExecutionChecks;
END_VAR
Check.IsTrue(ipSrcImage.IsValid, 'ipSrcImage must contain an image');
Check.IsTrue(ipSrcImage.IsPixelDepth(8), 'ipSrcImage must be 8 or 32 bit pixel depth');
Check.IsTrue((ipSrcImage.HasChannelCount(1) OR ipSrcImage.HasChannelCount(3)), 'ipSrcImage must contain 1 or 3 channels');

Check.IsTrue(ipTemplateImage.IsValid, 'ipTemplateImage must contain an image');
Check.IsTrue(ImagesHaveMatchingPixelFormats(ipSrcImage.Value, ipTemplateImage.Value), 'ipTemplateImage must have same pixel depth as ipSrcImage');
Check.IsTrue(ImagesHaveMatchingChannels(ipSrcImage.Value, ipTemplateImage.Value), 'ipTemplateImage must have same amount of channels as ipSrcImage');
Check.IsTrue(IsTemplateImageSmallerThanSourceImage(ipSrcImage.Value, ipTemplateImage.Value), 'ipTemplateImage must be smaller than ipSrcImage');
END_METHOD

END_FUNCTION_BLOCK

// Nodes/Image Analysis/Object Detection/Node_F_VN_MatchTemplateWalshExp
{attribute 'linkalways'} 
{attribute 'no_explicit_call' := 'This FB is a CLASS and must be accessed using methods or properties'}
{attribute 'enable_dynamic_creation'}
FUNCTION_BLOCK Node_F_VN_MatchTemplateWalshExp EXTENDS VisionNode
VAR
    ipSrcImage : _ITcVnImage;
    ipTemplateImage : _ITcVnImage;
	nProjections : _UDINT(10);
	eOptions : _ETcVnMatchTemplateWalshOptions(ETcVnMatchTemplateWalshOptions.TCVN_MTWO_NONE);
	nRotations : _UDINT(1);
    ipResultImage : _ITcVnImage;
    hrPrev : _HRESULT(S_OK);
	hresult : _HRESULT(S_OK);
END_VAR

METHOD FB_init : BOOL
VAR_INPUT
	bInitRetains : BOOL; // if TRUE, the retain variables are initialized (warm start / cold start)
	bInCopyCode : BOOL;  // if TRUE, the instance afterwards gets moved into the copy code (online change)
END_VAR
AddInput('ipSrcImage', ipSrcImage);
AddInput('ipTemplateImage', ipTemplateImage);
AddInput('nProjections', nProjections);
AddInput('eOptions', eOptions);
AddInput('nRotations', nRotations);
AddInput('hrPrev', hrPrev);
AddOutput('ipResultImage', ipResultImage);
AddOutput('hresult',hresult);
END_METHOD

METHOD PUBLIC  Clone : I_Node
VAR
	pNode : POINTER TO Node_F_VN_MatchTemplateWalshExp;
END_VAR
pNode := __NEW(Node_F_VN_MatchTemplateWalshExp);
Clone := pNode^;
END_METHOD

METHOD PROTECTED OnExecute
hresult.Value := F_VN_MatchTemplateWalshExp(
    ipSrcImage := ipSrcImage.Value,
    ipTemplateImage := ipTemplateImage.Value,
	ipResultImage := ipResultImage.Value,
	nProjections := nProjections.Value,
	eOptions := eOptions.Value,
	nRotations := nRotations.Value,	
	hrPrev:= hrPrev.Value);
END_METHOD

METHOD PUBLIC PreExecutionCheck
VAR_INPUT
	Check : I_PreExecutionChecks;
END_VAR
Check.IsTrue(ipSrcImage.IsValid, 'ipSrcImage must contain an image');
Check.IsTrue(ipSrcImage.IsPixelDepth(8), 'ipSrcImage must be 8 or 32 bit pixel depth');
Check.IsTrue((ipSrcImage.HasChannelCount(1) OR ipSrcImage.HasChannelCount(3)), 'ipSrcImage must contain 1 or 3 channels');

Check.IsTrue((nRotations.Value = 1 OR nRotations.Value = 2 OR nRotations.Value = 4), 'nRotations must be 1, 2 or 4');

Check.IsTrue(ipTemplateImage.IsValid, 'ipTemplateImage must contain an image');
Check.IsTrue(ImagesHaveMatchingPixelFormats(ipSrcImage.Value, ipTemplateImage.Value), 'ipTemplateImage must have same pixel depth as ipSrcImage');
Check.IsTrue(ImagesHaveMatchingChannels(ipSrcImage.Value, ipTemplateImage.Value), 'ipTemplateImage must have same amount of channels as ipSrcImage');
Check.IsTrue(IsTemplateImageSmallerThanSourceImage(ipSrcImage.Value, ipTemplateImage.Value), 'ipTemplateImage must be smaller than ipSrcImage');
END_METHOD

END_FUNCTION_BLOCK

// Nodes/Image Analysis/Object Detection/Node_F_VN_MergeRegions
{attribute 'linkalways'}
{attribute 'no_explicit_call' := 'This FB is a CLASS and must be accessed using methods or properties'}
{attribute 'enable_dynamic_creation'}
FUNCTION_BLOCK Node_F_VN_MergeRegions EXTENDS VisionNode
VAR
    ipSrcContainer : _ITcVnContainer;
    ipDestContainer : _ITcVnContainer;
    nDistance : _UDINT(0);
    nOptions : _ETcVnMergeRegionsOptions(ETcVnMergeRegionsOptions.TCVN_MRO_UPRIGHT_BOUNDING_RECT);
    hrPrev : _HRESULT(S_OK);
    hresult : _HRESULT(S_OK);
END_VAR

METHOD FB_init : BOOL
VAR_INPUT
    bInitRetains : BOOL;
    bInCopyCode : BOOL;
END_VAR
AddInput('ipSrcContainer', ipSrcContainer);
AddOutput('ipDestContainer', ipDestContainer);
AddParameter('nDistance', nDistance);
AddParameter('nOptions', nOptions);
AddInput('hrPrev', hrPrev);
AddOutput('hresult', hresult);
END_METHOD

METHOD PUBLIC Clone : I_Node
VAR
    pNode : POINTER TO Node_F_VN_MergeRegions;
END_VAR
pNode := __NEW(Node_F_VN_MergeRegions);
Clone := pNode^;
END_METHOD

METHOD PROTECTED OnExecute
hresult.Value := F_VN_MergeRegions(
    ipSrcContainer := ipSrcContainer.Value,
    ipDestContainer := ipDestContainer.Value,
    nDistance := nDistance.Value,
    nOptions := nOptions.Value,
    hrPrev := hrPrev.Value);
END_METHOD

METHOD PUBLIC PreExecutionCheck
VAR_INPUT
    Check : I_PreExecutionChecks;
END_VAR
Check.IsTrue(ipSrcContainer.IsValid, 'ipSrcContainer must contain a container');
Check.IsTrue(ipSrcContainer.IsType(TC_GLOBAL_CONST_LIST.ContainerType_Vector_TcVnRectangle_DINT), 'ipSrcContainer must contain TcVnRectangle_DINT elements');
Check.IsTrue(nOptions.Value = ETcVnMergeRegionsOptions.TCVN_MRO_UPRIGHT_BOUNDING_RECT, 'Unsupported region merge option');
END_METHOD

END_FUNCTION_BLOCK

// Nodes/Image Analysis/Object Detection/Node_F_VN_SalientFeatures
{attribute 'linkalways'}
{attribute 'no_explicit_call' := 'This FB is a CLASS and must be accessed using methods or properties'}
{attribute 'enable_dynamic_creation'}
FUNCTION_BLOCK Node_F_VN_SalientFeatures EXTENDS VisionNode
VAR
    ipSrcImage : _ITcVnImage;
    ipDestImage : _ITcVnImage;
    eMethod : _ETcVnSalientFeaturesMethod(ETcVnSalientFeaturesMethod.TCVN_SFM_WALSH_CODE);
    hrPrev : _HRESULT(S_OK);
    hresult : _HRESULT(S_OK);
END_VAR

METHOD FB_init : BOOL
VAR_INPUT
    bInitRetains : BOOL;
    bInCopyCode : BOOL;
END_VAR
AddInput('ipSrcImage', ipSrcImage);
AddOutput('ipDestImage', ipDestImage);
AddParameter('eMethod', eMethod);
AddInput('hrPrev', hrPrev);
AddOutput('hresult', hresult);
END_METHOD

METHOD PUBLIC Clone : I_Node
VAR
    pNode : POINTER TO Node_F_VN_SalientFeatures;
END_VAR
pNode := __NEW(Node_F_VN_SalientFeatures);
Clone := pNode^;
END_METHOD

METHOD PROTECTED OnExecute
hresult.Value := F_VN_SalientFeatures(
    ipSrcImage := ipSrcImage.Value,
    ipDestImage := ipDestImage.Value,
    eMethod := eMethod.Value,
    hrPrev := hrPrev.Value);
END_METHOD

METHOD PUBLIC PreExecutionCheck
VAR_INPUT
    Check : I_PreExecutionChecks;
END_VAR
Check.IsTrue(ipSrcImage.IsValid, 'ipSrcImage must contain an image');
Check.IsTrue(ipSrcImage.IsElementType(ETcVnElementType.TCVN_ET_USINT), 'ipSrcImage must contain USINT elements');
Check.IsTrue(ipSrcImage.HasChannelCount(1) OR ipSrcImage.HasChannelCount(3), 'ipSrcImage must contain 1 or 3 channels');
Check.IsTrue((eMethod.Value = ETcVnSalientFeaturesMethod.TCVN_SFM_WALSH_CODE) OR
             (eMethod.Value = ETcVnSalientFeaturesMethod.TCVN_SFM_SOBEL), 'Unsupported salient features method');
END_METHOD

END_FUNCTION_BLOCK

// Nodes/Image Analysis/Node_F_VN_CannyEdgeDetection
{attribute 'linkalways'} 
{attribute 'no_explicit_call' := 'This FB is a CLASS and must be accessed using methods or properties'}
{attribute 'enable_dynamic_creation'}
FUNCTION_BLOCK Node_F_VN_CannyEdgeDetection EXTENDS VisionNode
VAR
    ipSrcImage : _ITcVnImage;
    ipDestImage : _ITcVnImage;
    fThresholdLow : _LREAL(0.0);
    fThresholdHigh : _LREAL(0.0);
    hrPrev : _HRESULT(S_OK);
	hresult : _HRESULT(S_OK);
END_VAR

METHOD FB_init : BOOL
VAR_INPUT
	bInitRetains : BOOL; // if TRUE, the retain variables are initialized (warm start / cold start)
	bInCopyCode : BOOL;  // if TRUE, the instance afterwards gets moved into the copy code (online change)
END_VAR
AddInput('ipSrcImage', ipSrcImage);
AddParameter('fThresholdLow', fThresholdLow);
AddParameter('fThresholdHigh', fThresholdHigh);
AddInput('hrPrev', hrPrev);
AddOutput('ipDestImage', ipDestImage);
AddOutput('hresult', hresult);
END_METHOD

METHOD PUBLIC  Clone : I_Node
VAR
	pNode : POINTER TO Node_F_VN_CannyEdgeDetection;
END_VAR
pNode := __NEW(Node_F_VN_CannyEdgeDetection);
Clone := pNode^;
END_METHOD

METHOD PROTECTED OnExecute
hresult.Value := F_VN_CannyEdgeDetection(
	ipSrcImage := ipSrcImage.Value,
    ipDestImage := ipDestImage.Value,
    fThresholdLow := fThresholdLow.Value,
    fThresholdHigh := fThresholdHigh.Value,
	hrPrev:= hrPrev.Value);
END_METHOD

METHOD PUBLIC PreExecutionCheck
VAR_INPUT
	Check : I_PreExecutionChecks;
END_VAR
Check.IsTrue(ipSrcImage.IsValid, 'ipSrcImage must contain an image');
Check.IsTrue(ipSrcImage.IsPixelDepth(8), 'ipSrcImage must have 8 bit pixel depth');
END_METHOD

END_FUNCTION_BLOCK

// Nodes/Image Analysis/Node_F_VN_CannyEdgeDetectionExp
{attribute 'linkalways'} 
{attribute 'no_explicit_call' := 'This FB is a CLASS and must be accessed using methods or properties'}
{attribute 'enable_dynamic_creation'}
FUNCTION_BLOCK Node_F_VN_CannyEdgeDetectionExp EXTENDS VisionNode
VAR
    ipSrcImage : _ITcVnImage;
    ipDestImage : _ITcVnImage;
    fThresholdLow : _LREAL(0.0);
    fThresholdHigh : _LREAL(0.0);
    nApertureSize : _UDINT(3);
    bL2Gradient : _BOOL(FALSE);
    hrPrev : _HRESULT(S_OK);
	hresult : _HRESULT(S_OK);
END_VAR

METHOD FB_init : BOOL
VAR_INPUT
	bInitRetains : BOOL; // if TRUE, the retain variables are initialized (warm start / cold start)
	bInCopyCode : BOOL;  // if TRUE, the instance afterwards gets moved into the copy code (online change)
END_VAR
AddInput('ipSrcImage', ipSrcImage);
AddParameter('fThresholdLow', fThresholdLow);
AddParameter('fThresholdHigh', fThresholdHigh);
AddParameter('nApertureSize', nApertureSize);
AddParameter('bL2Gradient', bL2Gradient);
AddInput('hrPrev', hrPrev);
AddOutput('ipDestImage', ipDestImage);
AddOutput('hresult', hresult);
END_METHOD

METHOD PUBLIC  Clone : I_Node
VAR
	pNode : POINTER TO Node_F_VN_CannyEdgeDetectionExp;
END_VAR
pNode := __NEW(Node_F_VN_CannyEdgeDetectionExp);
Clone := pNode^;
END_METHOD

METHOD PROTECTED OnExecute
hresult.Value := F_VN_CannyEdgeDetectionExp(
	ipSrcImage := ipSrcImage.Value,
    ipDestImage := ipDestImage.Value,
    fThresholdLow := fThresholdLow.Value,
    fThresholdHigh := fThresholdHigh.Value,
    nApertureSize := nApertureSize.Value,
    bL2Gradient := bL2Gradient.Value,
	hrPrev:= hrPrev.Value);
END_METHOD

METHOD PUBLIC PreExecutionCheck
VAR_INPUT
	Check : I_PreExecutionChecks;
END_VAR
Check.IsTrue(ipSrcImage.IsValid, 'ipSrcImage must contain an image');
Check.IsTrue(ipSrcImage.IsPixelDepth(8), 'ipSrcImage must have 8 bit pixel depth');
Check.IsTrue(nApertureSize.Value >= 3, 'nApertureSize must be greater than or equal to 3');
Check.IsTrue(nApertureSize.IsOdd, 'nApertureSize must be an odd number');
END_METHOD

END_FUNCTION_BLOCK

// Nodes/Image Analysis/Node_F_VN_ConnectedComponents
{attribute 'linkalways'} 
{attribute 'no_explicit_call' := 'This FB is a CLASS and must be accessed using methods or properties'}
{attribute 'enable_dynamic_creation'}
FUNCTION_BLOCK Node_F_VN_ConnectedComponents EXTENDS VisionNode
VAR
    ipSrcImage : _ITcVnImage;
    ipLabelImage : _ITcVnImage;
    nLabels : _DINT(0);
    hrPrev : _HRESULT(S_OK);
	hresult : _HRESULT(S_OK);
END_VAR

METHOD FB_init : BOOL
VAR_INPUT
	bInitRetains : BOOL; // if TRUE, the retain variables are initialized (warm start / cold start)
	bInCopyCode : BOOL;  // if TRUE, the instance afterwards gets moved into the copy code (online change)
END_VAR
AddInput('ipSrcImage', ipSrcImage);
AddInput('hrPrev', hrPrev);
AddOutput('ipLabelImage', ipLabelImage);
AddOutput('nLabels', nLabels);
AddOutput('hresult', hresult);
END_METHOD

METHOD PUBLIC  Clone : I_Node
VAR
	pNode : POINTER TO Node_F_VN_ConnectedComponents;
END_VAR
pNode := __NEW(Node_F_VN_ConnectedComponents);
Clone := pNode^;
END_METHOD

METHOD PROTECTED OnExecute
hresult.Value := F_VN_ConnectedComponents(
	ipSrcImage := ipSrcImage.Value,
    ipLabelImage := ipLabelImage.Value,
    nLabels := nLabels.Value,
	hrPrev:= hrPrev.Value);
END_METHOD

METHOD PUBLIC PreExecutionCheck
VAR_INPUT
	Check : I_PreExecutionChecks;
END_VAR
Check.IsTrue(ipSrcImage.IsValid, 'ipSrcImage must contain an image');
Check.IsTrue(ipSrcImage.IsPixelDepth(8), 'ipSrcImage must be 8 bit pixel depth');
Check.IsTrue(ipSrcImage.HasChannelCount(1), 'ipSrcImage must contain 1 channel');
END_METHOD

END_FUNCTION_BLOCK

// Nodes/Image Analysis/Node_F_VN_ConnectedComponentsExp
{attribute 'linkalways'} 
{attribute 'no_explicit_call' := 'This FB is a CLASS and must be accessed using methods or properties'}
{attribute 'enable_dynamic_creation'}
FUNCTION_BLOCK Node_F_VN_ConnectedComponentsExp EXTENDS VisionNode
VAR
    ipSrcImage : _ITcVnImage;
    ipLabelImage : _ITcVnImage;
    nLabels : _DINT(0);
    eConnectivity : _ETcVnPixelConnectivity(ETcVnPixelConnectivity.TCVN_PC_4);
    eLabelType : _ETcVnElementType(ETcVnElementType.TCVN_ET_DINT);
    eAlgorithm : _ETcVnConnectedComponentsAlgorithm(ETcVnConnectedComponentsAlgorithm.TCVN_CCA_WU);
    hrPrev : _HRESULT(S_OK);
	hresult : _HRESULT(S_OK);
END_VAR

METHOD FB_init : BOOL
VAR_INPUT
	bInitRetains : BOOL; // if TRUE, the retain variables are initialized (warm start / cold start)
	bInCopyCode : BOOL;  // if TRUE, the instance afterwards gets moved into the copy code (online change)
END_VAR
AddInput('ipSrcImage', ipSrcImage);
AddParameter('eConnectivity', eConnectivity);
AddParameter('eLabelType', eLabelType);
AddParameter('eAlgorithm', eAlgorithm);
AddInput('hrPrev', hrPrev);
AddOutput('ipLabelImage', ipLabelImage);
AddOutput('nLabels', nLabels);
AddOutput('hresult', hresult);
END_METHOD

METHOD PUBLIC  Clone : I_Node
VAR
	pNode : POINTER TO Node_F_VN_ConnectedComponentsExp;
END_VAR
pNode := __NEW(Node_F_VN_ConnectedComponentsExp);
Clone := pNode^;
END_METHOD

METHOD PROTECTED OnExecute
hresult.Value := F_VN_ConnectedComponentsExp(
	ipSrcImage := ipSrcImage.Value,
    ipLabelImage := ipLabelImage.Value,
    nLabels := nLabels.Value,
    eConnectivity := eConnectivity.Value,
    eLabelType := eLabelType.Value,
    eAlgorithm := eAlgorithm.Value,
	hrPrev:= hrPrev.Value);
END_METHOD

METHOD PUBLIC PreExecutionCheck
VAR_INPUT
	Check : I_PreExecutionChecks;
END_VAR
Check.IsTrue(ipSrcImage.IsValid, 'ipSrcImage must contain an image');
Check.IsTrue(ipSrcImage.IsPixelDepth(8), 'ipSrcImage must be 8 bit pixel depth');
Check.IsTrue(ipSrcImage.HasChannelCount(1), 'ipSrcImage must contain 1 channel');
Check.IsTrue((eLabelType.Value = ETcVnElementType.TCVN_ET_DINT) OR
             (eLabelType.Value = ETcVnElementType.TCVN_ET_UINT), 'eLabelType must be DINT or UINT');
END_METHOD

END_FUNCTION_BLOCK

// Nodes/Image Analysis/Node_F_VN_ConnectedComponentsWithStats
{attribute 'linkalways'} 
{attribute 'no_explicit_call' := 'This FB is a CLASS and must be accessed using methods or properties'}
{attribute 'enable_dynamic_creation'}
FUNCTION_BLOCK Node_F_VN_ConnectedComponentsWithStats EXTENDS VisionNode
VAR
    ipSrcImage : _ITcVnImage;
    ipLabelImage : _ITcVnImage;
    ipBoundingBoxes : _ITcVnContainer;
    ipNumPixels : _ITcVnContainer;
    ipCentroids : _ITcVnContainer;
    nLabels : _DINT(0);
    hrPrev : _HRESULT(S_OK);
	hresult : _HRESULT(S_OK);
END_VAR

METHOD FB_init : BOOL
VAR_INPUT
	bInitRetains : BOOL; // if TRUE, the retain variables are initialized (warm start / cold start)
	bInCopyCode : BOOL;  // if TRUE, the instance afterwards gets moved into the copy code (online change)
END_VAR
AddInput('ipSrcImage', ipSrcImage);
AddInput('hrPrev', hrPrev);
AddOutput('ipLabelImage', ipLabelImage);
AddOutput('ipBoundingBoxes', ipBoundingBoxes);
AddOutput('ipNumPixels', ipNumPixels);
AddOutput('ipCentroids', ipCentroids);
AddOutput('nLabels', nLabels);
AddOutput('hresult', hresult);
END_METHOD

METHOD PUBLIC  Clone : I_Node
VAR
	pNode : POINTER TO Node_F_VN_ConnectedComponentsWithStats;
END_VAR
pNode := __NEW(Node_F_VN_ConnectedComponentsWithStats);
Clone := pNode^;
END_METHOD

METHOD PROTECTED OnExecute
hresult.Value := F_VN_ConnectedComponentsWithStats(
	ipSrcImage := ipSrcImage.Value,
    ipLabelImage := ipLabelImage.Value,
    ipBoundingBoxes := ipBoundingBoxes.Value,
    ipNumPixels := ipNumPixels.Value,
    ipCentroids := ipCentroids.Value,
    nLabels := nLabels.Value,
	hrPrev:= hrPrev.Value);
END_METHOD

METHOD PUBLIC PreExecutionCheck
VAR_INPUT
	Check : I_PreExecutionChecks;
END_VAR
Check.IsTrue(ipSrcImage.IsValid, 'ipSrcImage must contain an image');
Check.IsTrue(ipSrcImage.IsPixelDepth(8), 'ipSrcImage must be 8 bit pixel depth');
Check.IsTrue(ipSrcImage.HasChannelCount(1), 'ipSrcImage must contain 1 channel');
END_METHOD

END_FUNCTION_BLOCK

// Nodes/Image Analysis/Node_F_VN_ConnectedComponentsWithStatsExp
{attribute 'linkalways'} 
{attribute 'no_explicit_call' := 'This FB is a CLASS and must be accessed using methods or properties'}
{attribute 'enable_dynamic_creation'}
FUNCTION_BLOCK Node_F_VN_ConnectedComponentsWithStatsExp EXTENDS VisionNode
VAR
    ipSrcImage : _ITcVnImage;
    ipLabelImage : _ITcVnImage;
    ipBoundingBoxes : _ITcVnContainer;
    ipNumPixels : _ITcVnContainer;
    ipCentroids : _ITcVnContainer;
    nLabels : _DINT(0);
    eConnectivity : _ETcVnPixelConnectivity(ETcVnPixelConnectivity.TCVN_PC_4);
    eLabelType : _ETcVnElementType(ETcVnElementType.TCVN_ET_DINT);
    eAlgorithm : _ETcVnConnectedComponentsAlgorithm(ETcVnConnectedComponentsAlgorithm.TCVN_CCA_WU);
    hrPrev : _HRESULT(S_OK);
	hresult : _HRESULT(S_OK);
END_VAR

METHOD FB_init : BOOL
VAR_INPUT
	bInitRetains : BOOL; // if TRUE, the retain variables are initialized (warm start / cold start)
	bInCopyCode : BOOL;  // if TRUE, the instance afterwards gets moved into the copy code (online change)
END_VAR
AddInput('ipSrcImage', ipSrcImage);
AddParameter('eConnectivity', eConnectivity);
AddParameter('eLabelType', eLabelType);
AddParameter('eAlgorithm', eAlgorithm);
AddInput('hrPrev', hrPrev);
AddOutput('ipLabelImage', ipLabelImage);
AddOutput('nLabels', nLabels);
AddOutput('hresult', hresult);
END_METHOD

METHOD PUBLIC  Clone : I_Node
VAR
	pNode : POINTER TO Node_F_VN_ConnectedComponentsWithStatsExp;
END_VAR
pNode := __NEW(Node_F_VN_ConnectedComponentsWithStatsExp);
Clone := pNode^;
END_METHOD

METHOD PROTECTED OnExecute
hresult.Value := F_VN_ConnectedComponentsWithStatsExp(
	ipSrcImage := ipSrcImage.Value,
    ipLabelImage := ipLabelImage.Value,
    ipBoundingBoxes := ipBoundingBoxes.Value,
    ipNumPixels := ipNumPixels.Value,
    ipCentroids := ipCentroids.Value,
    nLabels := nLabels.Value,
    eConnectivity := eConnectivity.Value,
    eLabelType := eLabelType.Value,
    eAlgorithm := eAlgorithm.Value,
	hrPrev:= hrPrev.Value);
END_METHOD

METHOD PUBLIC PreExecutionCheck
VAR_INPUT
	Check : I_PreExecutionChecks;
END_VAR
Check.IsTrue(ipSrcImage.IsValid, 'ipSrcImage must contain an image');
Check.IsTrue(ipSrcImage.IsPixelDepth(8), 'ipSrcImage must be 8 bit pixel depth');
Check.IsTrue(ipSrcImage.HasChannelCount(1), 'ipSrcImage must contain 1 channel');
Check.IsTrue((eLabelType.Value = ETcVnElementType.TCVN_ET_DINT) OR
             (eLabelType.Value = ETcVnElementType.TCVN_ET_UINT), 'eLabelType must be DINT or UINT');
END_METHOD

END_FUNCTION_BLOCK

// Nodes/Image Analysis/Node_F_VN_CountNonZeroPixels
{attribute 'linkalways'} 
{attribute 'no_explicit_call' := 'This FB is a CLASS and must be accessed using methods or properties'}
{attribute 'enable_dynamic_creation'}
FUNCTION_BLOCK Node_F_VN_CountNonZeroPixels EXTENDS VisionNode
VAR
    ipSrcImage : _ITcVnImage;
    nNonZero : _ULINT(0);
    hrPrev : _HRESULT(S_OK);
	hresult : _HRESULT(S_OK);
END_VAR

METHOD FB_init : BOOL
VAR_INPUT
	bInitRetains : BOOL; // if TRUE, the retain variables are initialized (warm start / cold start)
	bInCopyCode : BOOL;  // if TRUE, the instance afterwards gets moved into the copy code (online change)
END_VAR
AddInput('ipSrcImage', ipSrcImage);
AddInput('hrPrev', hrPrev);
AddOutput('nNonZero', nNonZero);
AddOutput('hresult', hresult);
END_METHOD

METHOD PUBLIC  Clone : I_Node
VAR
	pNode : POINTER TO Node_F_VN_CountNonZeroPixels;
END_VAR
pNode := __NEW(Node_F_VN_CountNonZeroPixels);
Clone := pNode^;
END_METHOD

METHOD PROTECTED OnExecute
hresult.Value := F_VN_CountNonZeroPixels(
	ipSrcImage := ipSrcImage.Value,
    nNonZero := nNonZero.Value,
	hrPrev:= hrPrev.Value);
END_METHOD

METHOD PUBLIC PreExecutionCheck
VAR_INPUT
	Check : I_PreExecutionChecks;
END_VAR
Check.IsTrue(ipSrcImage.IsValid, 'ipSrcImage must contain an image');
Check.IsTrue(ipSrcImage.HasChannelCount(1), 'ipSrcImage must contain 1 channel');
END_METHOD

END_FUNCTION_BLOCK

// Nodes/Image Analysis/Node_F_VN_DistanceTransformation
{attribute 'linkalways'} 
{attribute 'no_explicit_call' := 'This FB is a CLASS and must be accessed using methods or properties'}
{attribute 'enable_dynamic_creation'}
FUNCTION_BLOCK Node_F_VN_DistanceTransformation EXTENDS VisionNode
VAR
    ipSrcImage : _ITcVnImage;
    ipDestImage : _ITcVnImage;
    eDistanceType : _ETcVnDistanceType(ETcVnDistanceType.TCVN_DT_L1);
    eMaskSize : _ETcVnDistanceTransformationMask(ETcVnDistanceTransformationMask.TCVN_DTM_PRECISE);
    hrPrev : _HRESULT(S_OK);
	hresult : _HRESULT(S_OK);
END_VAR

METHOD FB_init : BOOL
VAR_INPUT
	bInitRetains : BOOL; // if TRUE, the retain variables are initialized (warm start / cold start)
	bInCopyCode : BOOL;  // if TRUE, the instance afterwards gets moved into the copy code (online change)
END_VAR
AddInput('ipSrcImage', ipSrcImage);
AddParameter('eDistanceType', eDistanceType);
AddParameter('eMaskSize', eMaskSize);
AddInput('hrPrev', hrPrev);
AddOutput('ipDestImage', ipDestImage);
AddOutput('hresult',hresult);
END_METHOD

METHOD PUBLIC  Clone : I_Node
VAR
	pNode : POINTER TO Node_F_VN_DistanceTransformation;
END_VAR
pNode := __NEW(Node_F_VN_DistanceTransformation);
Clone := pNode^;
END_METHOD

METHOD PROTECTED OnExecute
hresult.Value := F_VN_DistanceTransformation(
    ipSrcImage := ipSrcImage.Value,
	ipDestImage := ipDestImage.Value,
    eDistanceType := eDistanceType.Value,
    eMaskSize := eMaskSize.Value,
	hrPrev:= hrPrev.Value);
END_METHOD

METHOD PUBLIC PreExecutionCheck
VAR_INPUT
	Check : I_PreExecutionChecks;
END_VAR
VAR
    distanceTypeIsValid : BOOL;
END_VAR
Check.IsTrue(ipSrcImage.IsValid, 'ipSrcImage must contain an image');
Check.IsTrue(ipSrcImage.HasChannelCount(1), 'ipSrcImage must have 1 channel');
Check.IsTrue(ipSrcImage.IsPixelDepth(8), 'ipSrcImage must have 8 bit pixel depth');

CASE eDistanceType.Value OF
    ETcVnDistanceType.TCVN_DT_L1,
    ETcVnDistanceType.TCVN_DT_L2,
    ETcVnDistanceType.TCVN_DT_C :
        distanceTypeIsValid := TRUE;
END_CASE
Check.IsTrue(distanceTypeIsValid, 'eDistanceType value is unsupported');
END_METHOD

END_FUNCTION_BLOCK

// Nodes/Image Analysis/Node_F_VN_DistanceTransformationExp
{attribute 'linkalways'} 
{attribute 'no_explicit_call' := 'This FB is a CLASS and must be accessed using methods or properties'}
{attribute 'enable_dynamic_creation'}
FUNCTION_BLOCK Node_F_VN_DistanceTransformationExp EXTENDS VisionNode
VAR
    ipSrcImage : _ITcVnImage;
    ipDestImage : _ITcVnImage;
    eDistanceType : _ETcVnDistanceType(ETcVnDistanceType.TCVN_DT_L1);
    eMaskSize : _ETcVnDistanceTransformationMask(ETcVnDistanceTransformationMask.TCVN_DTM_PRECISE);
    ipDestLabels : _ITcVnImage;
    eLabelType : _ETcVnDistanceTransformationLabel(ETcVnDistanceTransformationLabel.TCVN_DTL_CCOMP);
    hrPrev : _HRESULT(S_OK);
	hresult : _HRESULT(S_OK);
END_VAR

METHOD FB_init : BOOL
VAR_INPUT
	bInitRetains : BOOL; // if TRUE, the retain variables are initialized (warm start / cold start)
	bInCopyCode : BOOL;  // if TRUE, the instance afterwards gets moved into the copy code (online change)
END_VAR
AddInput('ipSrcImage', ipSrcImage);
AddParameter('eDistanceType', eDistanceType);
AddParameter('eMaskSize', eMaskSize);
AddParameter('eLabelType', eLabelType);
AddInput('hrPrev', hrPrev);
AddOutput('ipDestImage', ipDestImage);
AddOutput('ipDestLabels', ipDestLabels);
AddOutput('hresult',hresult);
END_METHOD

METHOD PUBLIC  Clone : I_Node
VAR
	pNode : POINTER TO Node_F_VN_DistanceTransformationExp;
END_VAR
pNode := __NEW(Node_F_VN_DistanceTransformationExp);
Clone := pNode^;
END_METHOD

METHOD PROTECTED OnExecute
hresult.Value := F_VN_DistanceTransformationExp(
    ipSrcImage := ipSrcImage.Value,
	ipDestImage := ipDestImage.Value,
    eDistanceType := eDistanceType.Value,
    eMaskSize := eMaskSize.Value,
    ipDestLabels := ipDestLabels.Value,
    eLabelType := eLabelType.Value,
	hrPrev:= hrPrev.Value);
END_METHOD

METHOD PUBLIC PreExecutionCheck
VAR_INPUT
	Check : I_PreExecutionChecks;
END_VAR
VAR
    distanceTypeIsValid : BOOL;
    maskSizeIsValid : BOOL;
END_VAR
Check.IsTrue(ipSrcImage.IsValid, 'ipSrcImage must contain an image');
Check.IsTrue(ipSrcImage.HasChannelCount(1), 'ipSrcImage must have 1 channel');
Check.IsTrue(ipSrcImage.IsPixelDepth(8), 'ipSrcImage must have 8 bit pixel depth');

CASE eDistanceType.Value OF
    ETcVnDistanceType.TCVN_DT_L1,
    ETcVnDistanceType.TCVN_DT_L2,
    ETcVnDistanceType.TCVN_DT_C :
        distanceTypeIsValid := TRUE;
END_CASE
Check.IsTrue(distanceTypeIsValid, 'eDistanceType value is unsupported');

CASE eMaskSize.Value OF
    ETcVnDistanceTransformationMask.TCVN_DTM_3,
    ETcVnDistanceTransformationMask.TCVN_DTM_5 :
        maskSizeIsValid := TRUE;
END_CASE
Check.IsTrue(maskSizeIsValid, 'maskSizeIsValid value is unsupported');
END_METHOD

END_FUNCTION_BLOCK

// Nodes/Image Analysis/Node_F_VN_GetConnectedComponent
{attribute 'linkalways'} 
{attribute 'no_explicit_call' := 'This FB is a CLASS and must be accessed using methods or properties'}
{attribute 'enable_dynamic_creation'}
FUNCTION_BLOCK Node_F_VN_GetConnectedComponent EXTENDS VisionNode
VAR
    ipLabelImage : _ITcVnImage;
    nLabelID : _DINT(0);
    ipMaskImage : _ITcVnImage;
    hrPrev : _HRESULT(S_OK);
	hresult : _HRESULT(S_OK);
END_VAR

METHOD FB_init : BOOL
VAR_INPUT
	bInitRetains : BOOL; // if TRUE, the retain variables are initialized (warm start / cold start)
	bInCopyCode : BOOL;  // if TRUE, the instance afterwards gets moved into the copy code (online change)
END_VAR
AddInput('ipLabelImage', ipLabelImage);
AddParameter('nLabelID', nLabelID);
AddInput('hrPrev', hrPrev);
AddOutput('ipMaskImage', ipMaskImage);
AddOutput('hresult', hresult);
END_METHOD

METHOD PUBLIC  Clone : I_Node
VAR
	pNode : POINTER TO Node_F_VN_GetConnectedComponent;
END_VAR
pNode := __NEW(Node_F_VN_GetConnectedComponent);
Clone := pNode^;
END_METHOD

METHOD PROTECTED OnExecute
hresult.Value := F_VN_GetConnectedComponent(
	ipLabelImage := ipLabelImage.Value,
    nLabelID := nLabelID.Value,
    ipMaskImage := ipMaskImage.Value,
	hrPrev:= hrPrev.Value);
END_METHOD

METHOD PUBLIC PreExecutionCheck
VAR_INPUT
	Check : I_PreExecutionChecks;
END_VAR
Check.IsTrue(ipLabelImage.IsValid, 'ipLabelImage must contain an image');
Check.IsTrue((ipLabelImage.IsPixelDepth(16)) OR (ipLabelImage.IsPixelDepth(32)), 'ipLabelImage must be 16 or 32 bit pixel depth');
Check.IsTrue(ipLabelImage.HasChannelCount(1), 'ipLabelImage must contain 1 channel');
END_METHOD

END_FUNCTION_BLOCK

// Nodes/Image Analysis/Node_F_VN_GetConnectedComponentExp
{attribute 'linkalways'} 
{attribute 'no_explicit_call' := 'This FB is a CLASS and must be accessed using methods or properties'}
{attribute 'enable_dynamic_creation'}
FUNCTION_BLOCK Node_F_VN_GetConnectedComponentExp EXTENDS VisionNode
VAR
    ipLabelImage : _ITcVnImage;
    nLabelID : _DINT(0);
    ipMaskImage : _ITcVnImage;
    ipContourPoints : _ITcVnContainer;
    hrPrev : _HRESULT(S_OK);
	hresult : _HRESULT(S_OK);
END_VAR

METHOD FB_init : BOOL
VAR_INPUT
	bInitRetains : BOOL; // if TRUE, the retain variables are initialized (warm start / cold start)
	bInCopyCode : BOOL;  // if TRUE, the instance afterwards gets moved into the copy code (online change)
END_VAR
AddInput('ipLabelImage', ipLabelImage);
AddParameter('nLabelID', nLabelID);
AddInput('hrPrev', hrPrev);
AddOutput('ipMaskImage', ipMaskImage);
AddOutput('ipContourPoints', ipContourPoints);
AddOutput('hresult', hresult);
END_METHOD

METHOD PUBLIC  Clone : I_Node
VAR
	pNode : POINTER TO Node_F_VN_GetConnectedComponentExp;
END_VAR
pNode := __NEW(Node_F_VN_GetConnectedComponentExp);
Clone := pNode^;
END_METHOD

METHOD PROTECTED OnExecute
hresult.Value := F_VN_GetConnectedComponentExp(
	ipLabelImage := ipLabelImage.Value,
    nLabelID := nLabelID.Value,
    ipMaskImage := ipMaskImage.Value,
    ipContourPoints := ipContourPoints.Value,
	hrPrev:= hrPrev.Value);
END_METHOD

METHOD PUBLIC PreExecutionCheck
VAR_INPUT
	Check : I_PreExecutionChecks;
END_VAR
Check.IsTrue(ipLabelImage.IsValid, 'ipLabelImage must contain an image');
Check.IsTrue((ipLabelImage.IsPixelDepth(16)) OR (ipLabelImage.IsPixelDepth(32)), 'ipLabelImage must be 16 or 32 bit pixel depth');
Check.IsTrue(ipLabelImage.HasChannelCount(1), 'ipLabelImage must contain 1 channel');
END_METHOD

END_FUNCTION_BLOCK

// Nodes/Image Analysis/Node_F_VN_ImageAbsoluteAverage
{attribute 'linkalways'} 
{attribute 'no_explicit_call' := 'This FB is a CLASS and must be accessed using methods or properties'}
{attribute 'enable_dynamic_creation'}
FUNCTION_BLOCK Node_F_VN_ImageAbsoluteAverage EXTENDS VisionNode
VAR
    ipSrcImage : _ITcVnImage;
    fAverage : _LREAL(0.0);
    hrPrev : _HRESULT(S_OK);
	hresult : _HRESULT(S_OK);
END_VAR

METHOD FB_init : BOOL
VAR_INPUT
	bInitRetains : BOOL; // if TRUE, the retain variables are initialized (warm start / cold start)
	bInCopyCode : BOOL;  // if TRUE, the instance afterwards gets moved into the copy code (online change)
END_VAR
AddInput('ipSrcImage', ipSrcImage);
AddInput('hrPrev', hrPrev);
AddOutput('fAverage', fAverage);
AddOutput('hresult', hresult);
END_METHOD

METHOD PUBLIC  Clone : I_Node
VAR
	pNode : POINTER TO Node_F_VN_ImageAbsoluteAverage;
END_VAR
pNode := __NEW(Node_F_VN_ImageAbsoluteAverage);
Clone := pNode^;
END_METHOD

METHOD PROTECTED OnExecute
hresult.Value := F_VN_ImageAbsoluteAverage(
	ipSrcImage := ipSrcImage.Value,
    fAverage := fAverage.Value,
	hrPrev:= hrPrev.Value);
END_METHOD

METHOD PUBLIC PreExecutionCheck
VAR_INPUT
	Check : I_PreExecutionChecks;
END_VAR
Check.IsTrue(ipSrcImage.IsValid, 'ipSrcImage must contain an image');
END_METHOD

END_FUNCTION_BLOCK

// Nodes/Image Analysis/Node_F_VN_ImageAverage
{attribute 'linkalways'} 
{attribute 'no_explicit_call' := 'This FB is a CLASS and must be accessed using methods or properties'}
{attribute 'enable_dynamic_creation'}
FUNCTION_BLOCK Node_F_VN_ImageAverage EXTENDS VisionNode
VAR
    ipSrcImage : _ITcVnImage;
    aAverage : _TcVnVector4_LREAL;
    hrPrev : _HRESULT(S_OK);
	hresult : _HRESULT(S_OK);
END_VAR

METHOD FB_init : BOOL
VAR_INPUT
	bInitRetains : BOOL; // if TRUE, the retain variables are initialized (warm start / cold start)
	bInCopyCode : BOOL;  // if TRUE, the instance afterwards gets moved into the copy code (online change)
END_VAR
AddInput('ipSrcImage', ipSrcImage);
AddInput('hrPrev', hrPrev);
AddOutput('aAverage', aAverage);
AddOutput('hresult', hresult);
END_METHOD

METHOD PUBLIC  Clone : I_Node
VAR
	pNode : POINTER TO Node_F_VN_ImageAverage;
END_VAR
pNode := __NEW(Node_F_VN_ImageAverage);
Clone := pNode^;
END_METHOD

METHOD PROTECTED OnExecute
hresult.Value := F_VN_ImageAverage(
	ipSrcImage := ipSrcImage.Value,
    aAverage := aAverage.Value,
	hrPrev:= hrPrev.Value);
END_METHOD

METHOD PUBLIC PreExecutionCheck
VAR_INPUT
	Check : I_PreExecutionChecks;
END_VAR
Check.IsTrue(ipSrcImage.IsValid, 'ipSrcImage must contain an image');
Check.IsTrue((ipSrcImage.HasChannelCount(1) OR
              ipSrcImage.HasChannelCount(2) OR
              ipSrcImage.HasChannelCount(3) OR
              ipSrcImage.HasChannelCount(4)), 'ipSrcImage must contain 1, 2, 3 or 4 channels');
END_METHOD

END_FUNCTION_BLOCK

// Nodes/Image Analysis/Node_F_VN_ImageAverageExp
{attribute 'linkalways'} 
{attribute 'no_explicit_call' := 'This FB is a CLASS and must be accessed using methods or properties'}
{attribute 'enable_dynamic_creation'}
FUNCTION_BLOCK Node_F_VN_ImageAverageExp EXTENDS VisionNode
VAR
    ipSrcImage : _ITcVnImage;
    aAverage : _TcVnVector4_LREAL;
    ipMask : _ITcVnImage;
    hrPrev : _HRESULT(S_OK);
	hresult : _HRESULT(S_OK);
END_VAR

METHOD FB_init : BOOL
VAR_INPUT
	bInitRetains : BOOL; // if TRUE, the retain variables are initialized (warm start / cold start)
	bInCopyCode : BOOL;  // if TRUE, the instance afterwards gets moved into the copy code (online change)
END_VAR
AddInput('ipSrcImage', ipSrcImage);
AddInput('ipMask', ipMask);
AddInput('hrPrev', hrPrev);
AddOutput('aAverage', aAverage);
AddOutput('hresult', hresult);
END_METHOD

METHOD PUBLIC  Clone : I_Node
VAR
	pNode : POINTER TO Node_F_VN_ImageAverageExp;
END_VAR
pNode := __NEW(Node_F_VN_ImageAverageExp);
Clone := pNode^;
END_METHOD

METHOD PROTECTED OnExecute
hresult.Value := F_VN_ImageAverageExp(
	ipSrcImage := ipSrcImage.Value,
    aAverage := aAverage.Value,
    ipMask := ipMask.Value,
	hrPrev:= hrPrev.Value);
END_METHOD

METHOD PUBLIC PreExecutionCheck
VAR_INPUT
	Check : I_PreExecutionChecks;
END_VAR
Check.IsTrue(ipSrcImage.IsValid, 'ipSrcImage must contain an image');
Check.IsTrue((ipSrcImage.HasChannelCount(1) OR
              ipSrcImage.HasChannelCount(2) OR
              ipSrcImage.HasChannelCount(3) OR
              ipSrcImage.HasChannelCount(4)), 'ipSrcImage must contain 1, 2, 3 or 4 channels');

Check.IsTrue(ipMask.IsValid, 'ipMask must contain an image');
Check.IsTrue(ipMask.HasChannelCount(1), 'ipMask must have 1 channel');
Check.IsTrue(ipMask.IsPixelDepth(8), 'ipMask must have 8 bit pixel depth');
Check.IsTrue(IsImage1SizeEqualToImage2Size(ipMask.Value, ipSrcImage.Value), 'ipMask must be the same size as ipSrcImage');
END_METHOD

END_FUNCTION_BLOCK

// Nodes/Image Analysis/Node_F_VN_ImageAverageStdDev
{attribute 'linkalways'} 
{attribute 'no_explicit_call' := 'This FB is a CLASS and must be accessed using methods or properties'}
{attribute 'enable_dynamic_creation'}
FUNCTION_BLOCK Node_F_VN_ImageAverageStdDev EXTENDS VisionNode
VAR
    ipSrcImage : _ITcVnImage;
    aAverage : _TcVnVector4_LREAL;
    aStdDev : _TcVnVector4_LREAL;
    hrPrev : _HRESULT(S_OK);
	hresult : _HRESULT(S_OK);
END_VAR

METHOD FB_init : BOOL
VAR_INPUT
	bInitRetains : BOOL; // if TRUE, the retain variables are initialized (warm start / cold start)
	bInCopyCode : BOOL;  // if TRUE, the instance afterwards gets moved into the copy code (online change)
END_VAR
AddInput('ipSrcImage', ipSrcImage);
AddInput('hrPrev', hrPrev);
AddOutput('aAverage', aAverage);
AddOutput('aStdDev', aStdDev);
AddOutput('hresult', hresult);
END_METHOD

METHOD PUBLIC  Clone : I_Node
VAR
	pNode : POINTER TO Node_F_VN_ImageAverageStdDev;
END_VAR
pNode := __NEW(Node_F_VN_ImageAverageStdDev);
Clone := pNode^;
END_METHOD

METHOD PROTECTED OnExecute
hresult.Value := F_VN_ImageAverageStdDev(
	ipSrcImage := ipSrcImage.Value,
    aAverage := aAverage.Value,
    aStdDev := aStdDev.Value,
	hrPrev:= hrPrev.Value);
END_METHOD

METHOD PUBLIC PreExecutionCheck
VAR_INPUT
	Check : I_PreExecutionChecks;
END_VAR
Check.IsTrue(ipSrcImage.IsValid, 'ipSrcImage must contain an image');
Check.IsTrue((ipSrcImage.HasChannelCount(1) OR
              ipSrcImage.HasChannelCount(2) OR
              ipSrcImage.HasChannelCount(3) OR
              ipSrcImage.HasChannelCount(4)), 'ipSrcImage must contain 1, 2, 3 or 4 channels');
END_METHOD

END_FUNCTION_BLOCK

// Nodes/Image Analysis/Node_F_VN_ImageAverageStdDevExp
{attribute 'linkalways'} 
{attribute 'no_explicit_call' := 'This FB is a CLASS and must be accessed using methods or properties'}
{attribute 'enable_dynamic_creation'}
FUNCTION_BLOCK Node_F_VN_ImageAverageStdDevExp EXTENDS VisionNode
VAR
    ipSrcImage : _ITcVnImage;
    aAverage : _TcVnVector4_LREAL;
    aStdDev : _TcVnVector4_LREAL;
    ipMask : _ITcVnImage;
    hrPrev : _HRESULT(S_OK);
	hresult : _HRESULT(S_OK);
END_VAR

METHOD FB_init : BOOL
VAR_INPUT
	bInitRetains : BOOL; // if TRUE, the retain variables are initialized (warm start / cold start)
	bInCopyCode : BOOL;  // if TRUE, the instance afterwards gets moved into the copy code (online change)
END_VAR
AddInput('ipSrcImage', ipSrcImage);
AddInput('ipMask', ipMask);
AddInput('hrPrev', hrPrev);
AddOutput('aAverage', aAverage);
AddOutput('aStdDev', aStdDev);
AddOutput('hresult', hresult);
END_METHOD

METHOD PUBLIC  Clone : I_Node
VAR
	pNode : POINTER TO Node_F_VN_ImageAverageStdDevExp;
END_VAR
pNode := __NEW(Node_F_VN_ImageAverageStdDevExp);
Clone := pNode^;
END_METHOD

METHOD PROTECTED OnExecute
hresult.Value := F_VN_ImageAverageStdDevExp(
	ipSrcImage := ipSrcImage.Value,
    aAverage := aAverage.Value,
    aStdDev := aStdDev.Value,
    ipMask := ipMask.Value,
	hrPrev:= hrPrev.Value);
END_METHOD

METHOD PUBLIC PreExecutionCheck
VAR_INPUT
	Check : I_PreExecutionChecks;
END_VAR
Check.IsTrue(ipSrcImage.IsValid, 'ipSrcImage must contain an image');
Check.IsTrue((ipSrcImage.HasChannelCount(1) OR
              ipSrcImage.HasChannelCount(2) OR
              ipSrcImage.HasChannelCount(3) OR
              ipSrcImage.HasChannelCount(4)), 'ipSrcImage must contain 1, 2, 3 or 4 channels');

Check.IsTrue(ipMask.IsValid, 'ipMask must contain an image');
Check.IsTrue(ipMask.HasChannelCount(1), 'ipMask must have 1 channel');
Check.IsTrue(ipMask.IsPixelDepth(8), 'ipMask must have 8 bit pixel depth');
Check.IsTrue(IsImage1SizeEqualToImage2Size(ipMask.Value, ipSrcImage.Value), 'ipMask must be the same size as ipSrcImage');
END_METHOD

END_FUNCTION_BLOCK

// Nodes/Image Analysis/Node_F_VN_ImageCenterOfMass
{attribute 'linkalways'} 
{attribute 'no_explicit_call' := 'This FB is a CLASS and must be accessed using methods or properties'}
{attribute 'enable_dynamic_creation'}
FUNCTION_BLOCK Node_F_VN_ImageCenterOfMass EXTENDS VisionNode
VAR
    ipSrcImage : _ITcVnImage;
    aCenterOfMass : _TcVnPoint2_LREAL;
    hrPrev : _HRESULT(S_OK);
	hresult : _HRESULT(S_OK);
END_VAR

METHOD FB_init : BOOL
VAR_INPUT
	bInitRetains : BOOL; // if TRUE, the retain variables are initialized (warm start / cold start)
	bInCopyCode : BOOL;  // if TRUE, the instance afterwards gets moved into the copy code (online change)
END_VAR
AddInput('ipSrcImage', ipSrcImage);
AddInput('hrPrev', hrPrev);
AddOutput('aCenterOfMass', aCenterOfMass);
AddOutput('hresult', hresult);
END_METHOD

METHOD PUBLIC  Clone : I_Node
VAR
	pNode : POINTER TO Node_F_VN_ImageCenterOfMass;
END_VAR
pNode := __NEW(Node_F_VN_ImageCenterOfMass);
Clone := pNode^;
END_METHOD

METHOD PROTECTED OnExecute
hresult.Value := F_VN_ImageCenterOfMass(
	ipSrcImage := ipSrcImage.Value,
    aCenterOfMass := aCenterOfMass.Value,
	hrPrev:= hrPrev.Value);
END_METHOD

METHOD PUBLIC PreExecutionCheck
VAR_INPUT
	Check : I_PreExecutionChecks;
END_VAR
Check.IsTrue(ipSrcImage.IsValid, 'ipSrcImage must contain an image');
Check.IsTrue(ipSrcImage.HasChannelCount(1), 'ipSrcImage must contain 1 channel');
END_METHOD

END_FUNCTION_BLOCK

// Nodes/Image Analysis/Node_F_VN_ImageCenterOfMassExp
{attribute 'linkalways'} 
{attribute 'no_explicit_call' := 'This FB is a CLASS and must be accessed using methods or properties'}
{attribute 'enable_dynamic_creation'}
FUNCTION_BLOCK Node_F_VN_ImageCenterOfMassExp EXTENDS VisionNode
VAR
    ipSrcImage : _ITcVnImage;
    aCenterOfMass : _TcVnPoint2_LREAL;
    ipMask : _ITcVnImage;
    hrPrev : _HRESULT(S_OK);
	hresult : _HRESULT(S_OK);
END_VAR

METHOD FB_init : BOOL
VAR_INPUT
	bInitRetains : BOOL; // if TRUE, the retain variables are initialized (warm start / cold start)
	bInCopyCode : BOOL;  // if TRUE, the instance afterwards gets moved into the copy code (online change)
END_VAR
AddInput('ipSrcImage', ipSrcImage);
AddInput('ipMask', ipMask);
AddInput('hrPrev', hrPrev);
AddOutput('aCenterOfMass', aCenterOfMass);
AddOutput('hresult', hresult);
END_METHOD

METHOD PUBLIC  Clone : I_Node
VAR
	pNode : POINTER TO Node_F_VN_ImageCenterOfMassExp;
END_VAR
pNode := __NEW(Node_F_VN_ImageCenterOfMassExp);
Clone := pNode^;
END_METHOD

METHOD PROTECTED OnExecute
hresult.Value := F_VN_ImageCenterOfMassExp(
	ipSrcImage := ipSrcImage.Value,
    aCenterOfMass := aCenterOfMass.Value,
    ipMask := ipMask.Value,
	hrPrev:= hrPrev.Value);
END_METHOD

METHOD PUBLIC PreExecutionCheck
VAR_INPUT
	Check : I_PreExecutionChecks;
END_VAR
Check.IsTrue(ipSrcImage.IsValid, 'ipSrcImage must contain an image');
Check.IsTrue(ipSrcImage.HasChannelCount(1), 'ipSrcImage must contain 1 channel');
Check.IsTrue(ipMask.IsValid, 'ipMask must contain an image');
Check.IsTrue(ipMask.HasChannelCount(1), 'ipMask must have 1 channel');
Check.IsTrue(ipMask.IsPixelDepth(8), 'ipMask must have 8 bit pixel depth');
Check.IsTrue(IsImage1SizeEqualToImage2Size(ipMask.Value, ipSrcImage.Value), 'ipMask must be the same size as ipSrcImage');
END_METHOD

END_FUNCTION_BLOCK

// Nodes/Image Analysis/Node_F_VN_ImageMedian
{attribute 'linkalways'} 
{attribute 'no_explicit_call' := 'This FB is a CLASS and must be accessed using methods or properties'}
{attribute 'enable_dynamic_creation'}
FUNCTION_BLOCK Node_F_VN_ImageMedian EXTENDS VisionNode
VAR
    ipSrcImage : _ITcVnImage;
    aMedian : _TcVnVector4_LREAL;
    hrPrev : _HRESULT(S_OK);
	hresult : _HRESULT(S_OK);
END_VAR

METHOD FB_init : BOOL
VAR_INPUT
	bInitRetains : BOOL; // if TRUE, the retain variables are initialized (warm start / cold start)
	bInCopyCode : BOOL;  // if TRUE, the instance afterwards gets moved into the copy code (online change)
END_VAR
AddInput('ipSrcImage', ipSrcImage);
AddInput('hrPrev', hrPrev);
AddOutput('aMedian', aMedian);
AddOutput('hresult', hresult);
END_METHOD

METHOD PUBLIC  Clone : I_Node
VAR
	pNode : POINTER TO Node_F_VN_ImageMedian;
END_VAR
pNode := __NEW(Node_F_VN_ImageMedian);
Clone := pNode^;
END_METHOD

METHOD PROTECTED OnExecute
hresult.Value := F_VN_ImageMedian(
	ipSrcImage := ipSrcImage.Value,
    aMedian := aMedian.Value,
	hrPrev:= hrPrev.Value);
END_METHOD

METHOD PUBLIC PreExecutionCheck
VAR_INPUT
	Check : I_PreExecutionChecks;
END_VAR
Check.IsTrue(ipSrcImage.IsValid, 'ipSrcImage must contain an image');
Check.IsTrue((ipSrcImage.HasChannelCount(1) OR
              ipSrcImage.HasChannelCount(2) OR
              ipSrcImage.HasChannelCount(3) OR
              ipSrcImage.HasChannelCount(4)), 'ipSrcImage must contain 1, 2, 3 or 4 channels');
END_METHOD

END_FUNCTION_BLOCK

// Nodes/Image Analysis/Node_F_VN_ImageMedianExp
{attribute 'linkalways'} 
{attribute 'no_explicit_call' := 'This FB is a CLASS and must be accessed using methods or properties'}
{attribute 'enable_dynamic_creation'}
FUNCTION_BLOCK Node_F_VN_ImageMedianExp EXTENDS VisionNode
VAR
    ipSrcImage : _ITcVnImage;
    aMedian : _TcVnVector4_LREAL;
    ipMask : _ITcVnImage;
    hrPrev : _HRESULT(S_OK);
	hresult : _HRESULT(S_OK);
END_VAR

METHOD FB_init : BOOL
VAR_INPUT
	bInitRetains : BOOL; // if TRUE, the retain variables are initialized (warm start / cold start)
	bInCopyCode : BOOL;  // if TRUE, the instance afterwards gets moved into the copy code (online change)
END_VAR
AddInput('ipSrcImage', ipSrcImage);
AddInput('ipMask', ipMask);
AddInput('hrPrev', hrPrev);
AddOutput('aMedian', aMedian);
AddOutput('hresult', hresult);
END_METHOD

METHOD PUBLIC  Clone : I_Node
VAR
	pNode : POINTER TO Node_F_VN_ImageMedianExp;
END_VAR
pNode := __NEW(Node_F_VN_ImageMedianExp);
Clone := pNode^;
END_METHOD

METHOD PROTECTED OnExecute
hresult.Value := F_VN_ImageMedianExp(
	ipSrcImage := ipSrcImage.Value,
    aMedian := aMedian.Value,
    ipMask := ipMask.Value,
	hrPrev:= hrPrev.Value);
END_METHOD

METHOD PUBLIC PreExecutionCheck
VAR_INPUT
	Check : I_PreExecutionChecks;
END_VAR
Check.IsTrue(ipSrcImage.IsValid, 'ipSrcImage must contain an image');
Check.IsTrue((ipSrcImage.HasChannelCount(1) OR
              ipSrcImage.HasChannelCount(2) OR
              ipSrcImage.HasChannelCount(3) OR
              ipSrcImage.HasChannelCount(4)), 'ipSrcImage must contain 1, 2, 3 or 4 channels');

Check.IsTrue(ipMask.IsValid, 'ipMask must contain an image');
Check.IsTrue(ipMask.HasChannelCount(1), 'ipMask must have 1 channel');
Check.IsTrue(ipMask.IsPixelDepth(8), 'ipMask must have 8 bit pixel depth');
Check.IsTrue(IsImage1SizeEqualToImage2Size(ipMask.Value, ipSrcImage.Value), 'ipMask must be the same size as ipSrcImage');
END_METHOD

END_FUNCTION_BLOCK

// Nodes/Image Analysis/Node_F_VN_ImageMoments
{attribute 'linkalways'} 
{attribute 'no_explicit_call' := 'This FB is a CLASS and must be accessed using methods or properties'}
{attribute 'enable_dynamic_creation'}
FUNCTION_BLOCK Node_F_VN_ImageMoments EXTENDS VisionNode
VAR
    ipImage : _ITcVnImage;
    stMoments : _TcVnMoments;
    bBinaryImage : _BOOL(FALSE);
    hrPrev : _HRESULT(S_OK);
	hresult : _HRESULT(S_OK);
END_VAR

METHOD FB_init : BOOL
VAR_INPUT
	bInitRetains : BOOL; // if TRUE, the retain variables are initialized (warm start / cold start)
	bInCopyCode : BOOL;  // if TRUE, the instance afterwards gets moved into the copy code (online change)
END_VAR
AddInput('ipImage', ipImage);
AddParameter('bBinaryImage', bBinaryImage);
AddInput('hrPrev', hrPrev);
AddOutput('stMoments', stMoments);
AddOutput('hresult', hresult);
END_METHOD

METHOD PUBLIC  Clone : I_Node
VAR
	pNode : POINTER TO Node_F_VN_ImageMoments;
END_VAR
pNode := __NEW(Node_F_VN_ImageMoments);
Clone := pNode^;
END_METHOD

METHOD PROTECTED OnExecute
hresult.Value := F_VN_ImageMoments(
	ipImage := ipImage.Value,
    stMoments := stMoments.Value,
    bBinaryImage := bBinaryImage.Value,
	hrPrev:= hrPrev.Value);
END_METHOD

METHOD PUBLIC PreExecutionCheck
VAR_INPUT
	Check : I_PreExecutionChecks;
END_VAR
Check.IsTrue(ipImage.IsValid, 'ipImage must contain an image');
Check.IsTrue(ipImage.HasChannelCount(1), 'ipImage must contain 1 channel');
Check.IsTrue((ipImage.IsPixelDepth(8) OR ipImage.IsPixelDepth(32)), 'ipImage must have 8 or 32 bit pixel depth');
END_METHOD

END_FUNCTION_BLOCK

// Nodes/Image Analysis/Node_F_VN_MaxPixelValue
{attribute 'linkalways'} 
{attribute 'no_explicit_call' := 'This FB is a CLASS and must be accessed using methods or properties'}
{attribute 'enable_dynamic_creation'}
FUNCTION_BLOCK Node_F_VN_MaxPixelValue EXTENDS VisionNode
VAR
    ipImage : _ITcVnImage;
    aMaxValue : _TcVnVector4_LREAL;
    aPosition : _TcVnPoint2_DINT;
    hrPrev : _HRESULT(S_OK);
	hresult : _HRESULT(S_OK);
END_VAR

METHOD FB_init : BOOL
VAR_INPUT
	bInitRetains : BOOL; // if TRUE, the retain variables are initialized (warm start / cold start)
	bInCopyCode : BOOL;  // if TRUE, the instance afterwards gets moved into the copy code (online change)
END_VAR
AddInput('ipImage', ipImage);
AddInput('hrPrev', hrPrev);
AddOutput('aMaxValue', aMaxValue);
AddOutput('aPosition', aPosition);
AddOutput('hresult', hresult);
END_METHOD

METHOD PUBLIC  Clone : I_Node
VAR
	pNode : POINTER TO Node_F_VN_MaxPixelValue;
END_VAR
pNode := __NEW(Node_F_VN_MaxPixelValue);
Clone := pNode^;
END_METHOD

METHOD PROTECTED OnExecute
hresult.Value := F_VN_MaxPixelValue(
	ipImage := ipImage.Value,
    aMaxValue := aMaxValue.Value,
    aPosition := aPosition.Value,
	hrPrev:= hrPrev.Value);
END_METHOD

METHOD PUBLIC PreExecutionCheck
VAR_INPUT
	Check : I_PreExecutionChecks;
END_VAR
Check.IsTrue(ipImage.IsValid, 'ipImage must contain an image');
Check.IsTrue((ipImage.HasChannelCount(1) OR
              ipImage.HasChannelCount(2) OR
              ipImage.HasChannelCount(3) OR
              ipImage.HasChannelCount(4)), 'ipImage must contain 1, 2, 3 or 4 channels');
END_METHOD

END_FUNCTION_BLOCK

// Nodes/Image Analysis/Node_F_VN_MaxPixelValueExp
{attribute 'linkalways'} 
{attribute 'no_explicit_call' := 'This FB is a CLASS and must be accessed using methods or properties'}
{attribute 'enable_dynamic_creation'}
FUNCTION_BLOCK Node_F_VN_MaxPixelValueExp EXTENDS VisionNode
VAR
    ipImage : _ITcVnImage;
    aMaxValue : _TcVnVector4_LREAL;
    aPosition : _TcVnPoint2_DINT;
    ipMask : _ITcVnImage;
    eVectorCompareMethod : _ETcVnVectorCompareMethod(ETcVnVectorCompareMethod.TCVN_VCM_EUCLIDEAN);
    hrPrev : _HRESULT(S_OK);
	hresult : _HRESULT(S_OK);
END_VAR

METHOD FB_init : BOOL
VAR_INPUT
	bInitRetains : BOOL; // if TRUE, the retain variables are initialized (warm start / cold start)
	bInCopyCode : BOOL;  // if TRUE, the instance afterwards gets moved into the copy code (online change)
END_VAR
AddInput('ipImage', ipImage);
AddInput('ipMask', ipMask);
AddParameter('eVectorCompareMethod', eVectorCompareMethod);
AddInput('hrPrev', hrPrev);
AddOutput('aMaxValue', aMaxValue);
AddOutput('aPosition', aPosition);
AddOutput('hresult', hresult);
END_METHOD

METHOD PUBLIC  Clone : I_Node
VAR
	pNode : POINTER TO Node_F_VN_MaxPixelValueExp;
END_VAR
pNode := __NEW(Node_F_VN_MaxPixelValueExp);
Clone := pNode^;
END_METHOD

METHOD PROTECTED OnExecute
hresult.Value := F_VN_MaxPixelValueExp(
	ipImage := ipImage.Value,
    aMaxValue := aMaxValue.Value,
    aPosition := aPosition.Value,
    ipMask := ipMask.Value,
    eVectorCompareMethod := eVectorCompareMethod.Value,
	hrPrev:= hrPrev.Value);
END_METHOD

METHOD PUBLIC PreExecutionCheck
VAR_INPUT
	Check : I_PreExecutionChecks;
END_VAR
Check.IsTrue(ipImage.IsValid, 'ipImage must contain an image');
Check.IsTrue((ipImage.HasChannelCount(1) OR
              ipImage.HasChannelCount(2) OR
              ipImage.HasChannelCount(3) OR
              ipImage.HasChannelCount(4)), 'ipImage must contain 1, 2, 3 or 4 channels');

// ipMask : Optional mask to specify which pixel positions are considered (USINT, set parameter to 0 if not required)
IF NOT IsValidImage(ipMask.Value) THEN
    RETURN;
END_IF

Check.IsTrue(ipMask.IsValid, 'ipMask must contain an image');
Check.IsTrue(ipMask.HasChannelCount(1), 'ipMask must have 1 channel');
Check.IsTrue(ipMask.IsPixelDepth(8), 'ipMask must have 8 bit pixel depth');
Check.IsTrue(IsImage1SizeEqualToImage2Size(ipMask.Value, ipImage.Value), 'ipMask must be the same size as ipImage');
END_METHOD

END_FUNCTION_BLOCK

// Nodes/Image Analysis/Node_F_VN_MinPixelValue
{attribute 'linkalways'} 
{attribute 'no_explicit_call' := 'This FB is a CLASS and must be accessed using methods or properties'}
{attribute 'enable_dynamic_creation'}
FUNCTION_BLOCK Node_F_VN_MinPixelValue EXTENDS VisionNode
VAR
    ipImage : _ITcVnImage;
    aMinValue : _TcVnVector4_LREAL;
    aPosition : _TcVnPoint2_DINT;
    hrPrev : _HRESULT(S_OK);
	hresult : _HRESULT(S_OK);
END_VAR

METHOD FB_init : BOOL
VAR_INPUT
	bInitRetains : BOOL; // if TRUE, the retain variables are initialized (warm start / cold start)
	bInCopyCode : BOOL;  // if TRUE, the instance afterwards gets moved into the copy code (online change)
END_VAR
AddInput('ipImage', ipImage);
AddInput('hrPrev', hrPrev);
AddOutput('aMinValue', aMinValue);
AddOutput('aPosition', aPosition);
AddOutput('hresult', hresult);
END_METHOD

METHOD PUBLIC  Clone : I_Node
VAR
	pNode : POINTER TO Node_F_VN_MinPixelValue;
END_VAR
pNode := __NEW(Node_F_VN_MinPixelValue);
Clone := pNode^;
END_METHOD

METHOD PROTECTED OnExecute
hresult.Value := F_VN_MinPixelValue(
	ipImage := ipImage.Value,
    aMinValue := aMinValue.Value,
    aPosition := aPosition.Value,
	hrPrev:= hrPrev.Value);
END_METHOD

METHOD PUBLIC PreExecutionCheck
VAR_INPUT
	Check : I_PreExecutionChecks;
END_VAR
Check.IsTrue(ipImage.IsValid, 'ipImage must contain an image');
Check.IsTrue((ipImage.HasChannelCount(1) OR
              ipImage.HasChannelCount(2) OR
              ipImage.HasChannelCount(3) OR
              ipImage.HasChannelCount(4)), 'ipImage must contain 1, 2, 3 or 4 channels');
END_METHOD

END_FUNCTION_BLOCK

// Nodes/Image Analysis/Node_F_VN_MinPixelValueExp
{attribute 'linkalways'} 
{attribute 'no_explicit_call' := 'This FB is a CLASS and must be accessed using methods or properties'}
{attribute 'enable_dynamic_creation'}
FUNCTION_BLOCK Node_F_VN_MinPixelValueExp EXTENDS VisionNode
VAR
    ipImage : _ITcVnImage;
    aMinValue : _TcVnVector4_LREAL;
    aPosition : _TcVnPoint2_DINT;
    ipMask : _ITcVnImage;
    eVectorCompareMethod : _ETcVnVectorCompareMethod(ETcVnVectorCompareMethod.TCVN_VCM_EUCLIDEAN);
    hrPrev : _HRESULT(S_OK);
	hresult : _HRESULT(S_OK);
END_VAR

METHOD FB_init : BOOL
VAR_INPUT
	bInitRetains : BOOL; // if TRUE, the retain variables are initialized (warm start / cold start)
	bInCopyCode : BOOL;  // if TRUE, the instance afterwards gets moved into the copy code (online change)
END_VAR
AddInput('ipImage', ipImage);
AddInput('ipMask', ipMask);
AddParameter('eVectorCompareMethod', eVectorCompareMethod);
AddInput('hrPrev', hrPrev);
AddOutput('aMinValue', aMinValue);
AddOutput('aPosition', aPosition);
AddOutput('hresult', hresult);
END_METHOD

METHOD PUBLIC  Clone : I_Node
VAR
	pNode : POINTER TO Node_F_VN_MinPixelValueExp;
END_VAR
pNode := __NEW(Node_F_VN_MinPixelValueExp);
Clone := pNode^;
END_METHOD

METHOD PROTECTED OnExecute
hresult.Value := F_VN_MinPixelValueExp(
	ipImage := ipImage.Value,
    aMinValue := aMinValue.Value,
    aPosition := aPosition.Value,
    ipMask := ipMask.Value,
    eVectorCompareMethod := eVectorCompareMethod.Value,
	hrPrev:= hrPrev.Value);
END_METHOD

METHOD PUBLIC PreExecutionCheck
VAR_INPUT
	Check : I_PreExecutionChecks;
END_VAR
Check.IsTrue(ipImage.IsValid, 'ipImage must contain an image');
Check.IsTrue((ipImage.HasChannelCount(1) OR
              ipImage.HasChannelCount(2) OR
              ipImage.HasChannelCount(3) OR
              ipImage.HasChannelCount(4)), 'ipImage must contain 1, 2, 3 or 4 channels');

// ipMask : Optional mask to specify which pixel positions are considered (USINT, set parameter to 0 if not required)
IF NOT IsValidImage(ipMask.Value) THEN
    RETURN;
END_IF

Check.IsTrue(ipMask.IsValid, 'ipMask must contain an image');
Check.IsTrue(ipMask.HasChannelCount(1), 'ipMask must have 1 channel');
Check.IsTrue(ipMask.IsPixelDepth(8), 'ipMask must have 8 bit pixel depth');
Check.IsTrue(IsImage1SizeEqualToImage2Size(ipMask.Value, ipImage.Value), 'ipMask must be the same size as ipImage');
END_METHOD

END_FUNCTION_BLOCK

// Nodes/Image Analysis/Node_F_VN_RegionOrientation
{attribute 'linkalways'} 
{attribute 'no_explicit_call' := 'This FB is a CLASS and must be accessed using methods or properties'}
{attribute 'enable_dynamic_creation'}
FUNCTION_BLOCK Node_F_VN_RegionOrientation EXTENDS VisionNode
VAR
    ipSrcImage : _ITcVnImage;
    stOrientation : _TcVnRotatedRectangle;
    hrPrev : _HRESULT(S_OK);
	hresult : _HRESULT(S_OK);
END_VAR

METHOD FB_init : BOOL
VAR_INPUT
	bInitRetains : BOOL; // if TRUE, the retain variables are initialized (warm start / cold start)
	bInCopyCode : BOOL;  // if TRUE, the instance afterwards gets moved into the copy code (online change)
END_VAR
AddInput('ipSrcImage', ipSrcImage);
AddInput('hrPrev', hrPrev);
AddOutput('stOrientation', stOrientation);
AddOutput('hresult', hresult);
END_METHOD

METHOD PUBLIC  Clone : I_Node
VAR
	pNode : POINTER TO Node_F_VN_RegionOrientation;
END_VAR
pNode := __NEW(Node_F_VN_RegionOrientation);
Clone := pNode^;
END_METHOD

METHOD PROTECTED OnExecute
hresult.Value := F_VN_RegionOrientation(
	ipSrcImage := ipSrcImage.Value,
    stOrientation := stOrientation.Value,
	hrPrev:= hrPrev.Value);
END_METHOD

METHOD PUBLIC PreExecutionCheck
VAR_INPUT
	Check : I_PreExecutionChecks;
END_VAR
Check.IsTrue(ipSrcImage.IsValid, 'ipSrcImage must contain an image');
Check.IsTrue(ipSrcImage.HasChannelCount(1), 'ipSrcImage must contain 1 channel');
END_METHOD

END_FUNCTION_BLOCK

// Nodes/Image Analysis/Node_F_VN_RegionOrientationExp
{attribute 'linkalways'} 
{attribute 'no_explicit_call' := 'This FB is a CLASS and must be accessed using methods or properties'}
{attribute 'enable_dynamic_creation'}
FUNCTION_BLOCK Node_F_VN_RegionOrientationExp EXTENDS VisionNode
VAR
    ipSrcImage : _ITcVnImage;
    stOrientation : _TcVnRotatedRectangle;
    eMethod : _ETcVnOrientationMethod(ETcVnOrientationMethod.TCVN_OM_PCA);
    hrPrev : _HRESULT(S_OK);
	hresult : _HRESULT(S_OK);
END_VAR

METHOD FB_init : BOOL
VAR_INPUT
	bInitRetains : BOOL; // if TRUE, the retain variables are initialized (warm start / cold start)
	bInCopyCode : BOOL;  // if TRUE, the instance afterwards gets moved into the copy code (online change)
END_VAR
AddInput('ipSrcImage', ipSrcImage);
AddParameter('eMethod', eMethod);
AddInput('hrPrev', hrPrev);
AddOutput('stOrientation', stOrientation);
AddOutput('hresult', hresult);
END_METHOD

METHOD PUBLIC  Clone : I_Node
VAR
	pNode : POINTER TO Node_F_VN_RegionOrientationExp;
END_VAR
pNode := __NEW(Node_F_VN_RegionOrientationExp);
Clone := pNode^;
END_METHOD

METHOD PROTECTED OnExecute
hresult.Value := F_VN_RegionOrientationExp(
	ipSrcImage := ipSrcImage.Value,
    stOrientation := stOrientation.Value,
    eMethod := eMethod.Value,
	hrPrev:= hrPrev.Value);
END_METHOD

METHOD PUBLIC PreExecutionCheck
VAR_INPUT
	Check : I_PreExecutionChecks;
END_VAR
Check.IsTrue(ipSrcImage.IsValid, 'ipSrcImage must contain an image');
Check.IsTrue(ipSrcImage.HasChannelCount(1), 'ipSrcImage must contain 1 channel');
END_METHOD

END_FUNCTION_BLOCK

// Nodes/Image Analysis/Node_F_VN_UprightInnerRectangle
{attribute 'linkalways'} 
{attribute 'no_explicit_call' := 'This FB is a CLASS and must be accessed using methods or properties'}
{attribute 'enable_dynamic_creation'}
FUNCTION_BLOCK Node_F_VN_UprightInnerRectangle EXTENDS VisionNode
VAR
    ipSrcImage : _ITcVnImage;
    stRectangle : _TcVnRectangle_DINT;
    hrPrev : _HRESULT(S_OK);
	hresult : _HRESULT(S_OK);
END_VAR

METHOD FB_init : BOOL
VAR_INPUT
	bInitRetains : BOOL; // if TRUE, the retain variables are initialized (warm start / cold start)
	bInCopyCode : BOOL;  // if TRUE, the instance afterwards gets moved into the copy code (online change)
END_VAR
AddInput('ipSrcImage', ipSrcImage);
AddInput('hrPrev', hrPrev);
AddOutput('stRectangle', stRectangle);
AddOutput('hresult', hresult);
END_METHOD

METHOD PUBLIC  Clone : I_Node
VAR
	pNode : POINTER TO Node_F_VN_UprightInnerRectangle;
END_VAR
pNode := __NEW(Node_F_VN_UprightInnerRectangle);
Clone := pNode^;
END_METHOD

METHOD PROTECTED OnExecute
hresult.Value := F_VN_UprightInnerRectangle(
	ipSrcImage := ipSrcImage.Value,
    stRectangle := stRectangle.Value,
	hrPrev:= hrPrev.Value);
END_METHOD

METHOD PUBLIC PreExecutionCheck
VAR_INPUT
	Check : I_PreExecutionChecks;
END_VAR
Check.IsTrue(ipSrcImage.IsValid, 'ipSrcImage must contain an image');
Check.IsTrue(ipSrcImage.IsPixelDepth(8), 'ipSrcImage must be 8 bit pixel depth');
Check.IsTrue(ipSrcImage.HasChannelCount(1), 'ipSrcImage must contain 1 channel');
END_METHOD

END_FUNCTION_BLOCK

// Nodes/Image Analysis/Node_F_VN_UprightInnerRectangleExp
{attribute 'linkalways'} 
{attribute 'no_explicit_call' := 'This FB is a CLASS and must be accessed using methods or properties'}
{attribute 'enable_dynamic_creation'}
FUNCTION_BLOCK Node_F_VN_UprightInnerRectangleExp EXTENDS VisionNode
VAR
    ipSrcImage : _ITcVnImage;
    stRectangle : _TcVnRectangle_DINT;
    nDownScaleFactor : _DINT(-1);
    hrPrev : _HRESULT(S_OK);
	hresult : _HRESULT(S_OK);
END_VAR

METHOD FB_init : BOOL
VAR_INPUT
	bInitRetains : BOOL; // if TRUE, the retain variables are initialized (warm start / cold start)
	bInCopyCode : BOOL;  // if TRUE, the instance afterwards gets moved into the copy code (online change)
END_VAR
AddInput('ipSrcImage', ipSrcImage);
AddParameter('nDownScaleFactor', nDownScaleFactor);
AddInput('hrPrev', hrPrev);
AddOutput('stRectangle', stRectangle);
AddOutput('hresult', hresult);
END_METHOD

METHOD PUBLIC  Clone : I_Node
VAR
	pNode : POINTER TO Node_F_VN_UprightInnerRectangleExp;
END_VAR
pNode := __NEW(Node_F_VN_UprightInnerRectangleExp);
Clone := pNode^;
END_METHOD

METHOD PROTECTED OnExecute
hresult.Value := F_VN_UprightInnerRectangleExp(
	ipSrcImage := ipSrcImage.Value,
    stRectangle := stRectangle.Value,
    nDownScaleFactor := nDownScaleFactor.Value,
	hrPrev:= hrPrev.Value);
END_METHOD

METHOD PUBLIC PreExecutionCheck
VAR_INPUT
	Check : I_PreExecutionChecks;
END_VAR
Check.IsTrue(ipSrcImage.IsValid, 'ipSrcImage must contain an image');
Check.IsTrue(ipSrcImage.IsPixelDepth(8), 'ipSrcImage must be 8 bit pixel depth');
Check.IsTrue(ipSrcImage.HasChannelCount(1), 'ipSrcImage must contain 1 channel');
Check.IsTrue(nDownScaleFactor.Value >= -1, 'nDownScaleFactor must be greater than or equal to -1');
END_METHOD

END_FUNCTION_BLOCK

// Nodes/Image Color and Contrast Processing/Node_F_VN_ApplyColorMap
{attribute 'linkalways'} 
{attribute 'no_explicit_call' := 'This FB is a CLASS and must be accessed using methods or properties'}
{attribute 'enable_dynamic_creation'}
FUNCTION_BLOCK Node_F_VN_ApplyColorMap EXTENDS VisionNode
VAR
	ipSrcImage : _ITcVnImage;
    ipDestImage : _ITcVnImage;
    ipColorMap : _ITcVnContainer;
    hrPrev : _HRESULT(S_OK);
	hresult : _HRESULT(S_OK);
END_VAR

METHOD FB_init : BOOL
VAR_INPUT
	bInitRetains : BOOL; // if TRUE, the retain variables are initialized (warm start / cold start)
	bInCopyCode : BOOL;  // if TRUE, the instance afterwards gets moved into the copy code (online change)
END_VAR
AddInput('ipSrcImage', ipSrcImage);
AddInput('ipColorMap', ipColorMap);
AddInput('hrPrev', hrPrev);
AddOutput('ipDestImage', ipDestImage);
AddOutput('hresult',hresult);
END_METHOD

METHOD PUBLIC  Clone : I_Node
VAR
	pNode : POINTER TO Node_F_VN_ApplyColorMap;
END_VAR
pNode := __NEW(Node_F_VN_ApplyColorMap);
Clone := pNode^;
END_METHOD

METHOD PROTECTED OnExecute
hresult.Value := F_VN_ApplyColorMap(
	ipSrcImage   := ipSrcImage.Value,
    ipDestImage   := ipDestImage.Value,
	ipColorMap := ipColorMap.Value,
	hrPrev := hrPrev.Value);
END_METHOD

METHOD PUBLIC PreExecutionCheck
VAR_INPUT
	Check : I_PreExecutionChecks;
END_VAR
VAR
    colorMapSize : ULINT;
END_VAR
Check.IsTrue(ipSrcImage.IsValid, 'ipSrcImage must contain an image');
Check.IsTrue(ipSrcImage.HasChannelCount(1), 'ipSrcImage must have 1 channel');

Check.IsTrue(ipColorMap.IsValid, 'ipColorMap must be a valid container');
Check.IsTrue(ipColorMap.IsType(TC_GLOBAL_CONST_LIST.ContainerType_Vector_TcVnVector3_REAL), 'ipColorMap contains incorrect type');

F_VN_GetNumberOfElements(ipColorMap.Value, colorMapSize, S_OK);

CASE colorMapSize OF
    256 :
        Check.IsTrue(ipSrcImage.IsPixelDepth(8), 'ipSrcImage must have 8 bit pixel depth');
    65536 :
        Check.IsTrue(ipSrcImage.IsPixelDepth(16), 'ipSrcImage must have 16 bit pixel depth');
ELSE
    Check.Fail('ipColorMp must contain 256 or 65536 elements');
END_CASE
END_METHOD

END_FUNCTION_BLOCK

// Nodes/Image Color and Contrast Processing/Node_F_VN_Clahe
{attribute 'linkalways'} 
{attribute 'no_explicit_call' := 'This FB is a CLASS and must be accessed using methods or properties'}
{attribute 'enable_dynamic_creation'}
FUNCTION_BLOCK Node_F_VN_Clahe EXTENDS VisionNode
VAR
	ipSrcImage : _ITcVnImage;
    ipDestImage : _ITcVnImage;
    hrPrev : _HRESULT(S_OK);
	hresult : _HRESULT(S_OK);
END_VAR

METHOD FB_init : BOOL
VAR_INPUT
	bInitRetains : BOOL; // if TRUE, the retain variables are initialized (warm start / cold start)
	bInCopyCode : BOOL;  // if TRUE, the instance afterwards gets moved into the copy code (online change)
END_VAR
AddInput('ipSrcImage', ipSrcImage);
AddInput('hrPrev', hrPrev);
AddOutput('ipDestImage', ipDestImage);
AddOutput('hresult',hresult);
END_METHOD

METHOD PUBLIC  Clone : I_Node
VAR
	pNode : POINTER TO Node_F_VN_Clahe;
END_VAR
pNode := __NEW(Node_F_VN_Clahe);
Clone := pNode^;
END_METHOD

METHOD PROTECTED OnExecute
hresult.Value := F_VN_Clahe(
	ipSrcImage := ipSrcImage.Value,
    ipDestImage := ipDestImage.Value,
	hrPrev := hrPrev.Value);
END_METHOD

METHOD PUBLIC PreExecutionCheck
VAR_INPUT
	Check : I_PreExecutionChecks;
END_VAR
VAR
    colorMapSize : ULINT;
END_VAR
Check.IsTrue(ipSrcImage.IsValid, 'ipSrcImage must contain an image');
Check.IsTrue(ipSrcImage.HasChannelCount(1), 'ipSrcImage must have 1 channel');
Check.IsTrue((ipSrcImage.IsPixelDepth(8) OR
              ipSrcImage.IsPixelDepth(16)), 'ipSrcImage must have 8 or 16 bit pixel depth');
END_METHOD

END_FUNCTION_BLOCK

// Nodes/Image Color and Contrast Processing/Node_F_VN_ClaheExp
{attribute 'linkalways'} 
{attribute 'no_explicit_call' := 'This FB is a CLASS and must be accessed using methods or properties'}
{attribute 'enable_dynamic_creation'}
FUNCTION_BLOCK Node_F_VN_ClaheExp EXTENDS VisionNode
VAR
	ipSrcImage : _ITcVnImage;
    ipDestImage : _ITcVnImage;
    fClipLimit  : _LREAL(0.0);
    nTilesX     : _UDINT(0);
    nTilesY     : _UDINT(0);
    hrPrev : _HRESULT(S_OK);
	hresult : _HRESULT(S_OK);
END_VAR

METHOD FB_init : BOOL
VAR_INPUT
	bInitRetains : BOOL; // if TRUE, the retain variables are initialized (warm start / cold start)
	bInCopyCode : BOOL;  // if TRUE, the instance afterwards gets moved into the copy code (online change)
END_VAR
AddInput('ipSrcImage', ipSrcImage);
AddParameter('fClipLimit', fClipLimit);
AddParameter('nTilesX', nTilesX);
AddParameter('nTilesY', nTilesY);
AddInput('hrPrev', hrPrev);
AddOutput('ipDestImage', ipDestImage);
AddOutput('hresult',hresult);
END_METHOD

METHOD PUBLIC  Clone : I_Node
VAR
	pNode : POINTER TO Node_F_VN_ClaheExp;
END_VAR
pNode := __NEW(Node_F_VN_ClaheExp);
Clone := pNode^;
END_METHOD

METHOD PROTECTED OnExecute
hresult.Value := F_VN_ClaheExp(
	ipSrcImage := ipSrcImage.Value,
    fClipLimit := fClipLimit.Value,
    nTilesX := nTilesX.Value,
    nTilesY := nTilesY.Value,
    ipDestImage   := ipDestImage.Value,
	hrPrev := hrPrev.Value);
END_METHOD

METHOD PUBLIC PreExecutionCheck
VAR_INPUT
	Check : I_PreExecutionChecks;
END_VAR
VAR
    colorMapSize : ULINT;
END_VAR
Check.IsTrue(ipSrcImage.IsValid, 'ipSrcImage must contain an image');
Check.IsTrue(ipSrcImage.HasChannelCount(1), 'ipSrcImage must have 1 channel');
Check.IsTrue((ipSrcImage.IsPixelDepth(8) OR
              ipSrcImage.IsPixelDepth(16)), 'ipSrcImage must have 8 or 16 bit pixel depth');
END_METHOD

END_FUNCTION_BLOCK

// Nodes/Image Color and Contrast Processing/Node_F_VN_ConvertColorSpace
{attribute 'linkalways'} 
{attribute 'no_explicit_call' := 'This FB is a CLASS and must be accessed using methods or properties'}
{attribute 'enable_dynamic_creation'}
FUNCTION_BLOCK Node_F_VN_ConvertColorSpace EXTENDS VisionNode
VAR
	ipSrcImage : _ITcVnImage;
    ipDestImage : _ITcVnImage;
    eTransform : _ETcVnColorSpaceTransform(ETcVnColorSpaceTransform.TCVN_CST_RGBA_TO_GRAY);
    hrPrev : _HRESULT(S_OK);
	hresult : _HRESULT(S_OK);
END_VAR

METHOD FB_init : BOOL
VAR_INPUT
	bInitRetains : BOOL; // if TRUE, the retain variables are initialized (warm start / cold start)
	bInCopyCode : BOOL;  // if TRUE, the instance afterwards gets moved into the copy code (online change)
END_VAR
AddInput('ipSrcImage', ipSrcImage);
AddInput('hrPrev', hrPrev);
AddOutput('ipDestImage', ipDestImage);
AddOutput('hresult',hresult);
AddParameter('eTransform', eTransform);
END_METHOD

METHOD PUBLIC  Clone : I_Node
VAR
	pNode : POINTER TO Node_F_VN_ConvertColorSpace;
END_VAR
pNode := __NEW(Node_F_VN_ConvertColorSpace);
Clone := pNode^;
END_METHOD

METHOD PROTECTED OnExecute
hresult.Value := F_VN_ConvertColorSpace(
	ipSrcImage   := ipSrcImage.Value, 
	ipDestImage:= ipDestImage.Value, 
	eTransform := eTransform.Value, 
	hrPrev := hrPrev.Value);
END_METHOD

